LIN {X 0,Y 287.709,Z 666.106,A -85,B 0,C 180,E1 12553.998,E2 12553.998} C_VEL
LIN {X 0,Y 281.324,Z 683.017,A -85,B 0,C 180,E1 12550.975,E2 12550.975} C_VEL
LIN {X 0,Y 275.503,Z 697.991,A -85,B 0,C 180,E1 12547.706,E2 12547.706} C_VEL
LIN {X 0,Y 269.962,Z 712.115,A -85,B 0,C 180,E1 12543.941,E2 12543.941} C_VEL
LIN {X 0,Y 265.266,Z 724.533,A -85,B 0,C 180,E1 12539.897,E2 12539.897} C_VEL
LIN {X 0,Y 261.375,Z 735.692,A -85,B 0,C 180,E1 12535.368,E2 12535.368} C_VEL
LIN {X 0,Y 258.724,Z 744.628,A -85,B 0,C 180,E1 12530.826,E2 12530.826} C_VEL
LIN {X 0,Y 257.127,Z 751.706,A -85,B 0,C 180,E1 12526.164,E2 12526.164} C_VEL
LIN {X 0,Y 256.425,Z 757.033,A -85,B 0,C 180,E1 12521.47,E2 12521.47} C_VEL
LIN {X 0,Y 256.333,Z 760.365,A -85,B 0,C 180,E1 12517.17,E2 12517.17} C_VEL
LIN {X 0,Y 256.431,Z 762.152,A -85,B 0,C 180,E1 12513.129,E2 12513.129} C_VEL
LIN {X 0,Y 256.464,Z 762.649,A -85,B 0,C 180,E1 12509.106,E2 12509.106} C_VEL
LIN {X 0,Y 256.359,Z 761.883,A -85,B 0,C 180,E1 12505.077,E2 12505.077} C_VEL
LIN {X 0,Y 256.284,Z 759.711,A -85,B 0,C 180,E1 12500.764,E2 12500.764} C_VEL
LIN {X 0,Y 256.66,Z 755.693,A -85,B 0,C 180,E1 12496.023,E2 12496.023} C_VEL
LIN {X 0,Y 257.964,Z 749.671,A -85,B 0,C 180,E1 12491.036,E2 12491.036} C_VEL
LIN {X 0,Y 260.411,Z 741.966,A -85,B 0,C 180,E1 12486.224,E2 12486.224} C_VEL
LIN {X 0,Y 264.156,Z 732.301,A -85,B 0,C 180,E1 12481.515,E2 12481.515} C_VEL
LIN {X 0,Y 269.345,Z 720.5,A -85,B 0,C 180,E1 12476.928,E2 12476.928} C_VEL
LIN {X 0,Y 275.298,Z 707.685,A -85,B 0,C 180,E1 12472.922,E2 12472.922} C_VEL
LIN {X 0,Y 282.458,Z 692.507,A -85,B 0,C 180,E1 12469.09,E2 12469.09} C_VEL
LIN {X 0,Y 289.833,Z 676.554,A -85,B 0,C 180,E1 12465.824,E2 12465.824} C_VEL
LIN {X 0,Y 297.598,Z 658.888,A -85,B 0,C 180,E1 12462.909,E2 12462.909} C_VEL
LIN {X 0,Y 305.008,Z 640.783,A -85,B 0,C 180,E1 12460.488,E2 12460.488} C_VEL
LIN {X 0,Y 312.373,Z 620.899,A -85,B 0,C 180,E1 12458.352,E2 12458.352} C_VEL
LIN {X 0,Y 318.941,Z 600.695,A -85,B 0,C 180,E1 12456.626,E2 12456.626} C_VEL
LIN {X 0,Y 321.995,Z 590.5,A -85,B 0,C 180,E1 12455.859,E2 12455.859} C_VEL
LIN {X 0,Y 315.93,Z 596.748,A -85,B 0,C 180,E1 12455.169,E2 12455.169} C_VEL
LIN {X 0,Y 312.395,Z 600.249,A -85,B 0,C 180,E1 12454.729,E2 12454.729} C_VEL
LIN {X 0,Y 306.375,Z 605.854,A -85,B 0,C 180,E1 12453.921,E2 12453.921} C_VEL
LIN {X 0,Y 302.961,Z 608.865,A -85,B 0,C 180,E1 12453.445,E2 12453.445} C_VEL
LIN {X 0,Y 298.097,Z 612.903,A -85,B 0,C 180,E1 12452.684,E2 12452.684} C_VEL
LIN {X 0,Y 295.592,Z 614.826,A -85,B 0,C 180,E1 12452.259,E2 12452.259} C_VEL
LIN {X 0,Y 291.07,Z 618.329,A -85,B 0,C 180,E1 12451.475,E2 12451.475} C_VEL
LIN {X 0,Y 289.437,Z 619.438,A -85,B 0,C 180,E1 12451.094,E2 12451.094} C_VEL
LIN {X 0,Y 284.898,Z 632.295,A -85,B 0,C 180,E1 12448.737,E2 12448.737} C_VEL
LIN {X 0,Y 280.252,Z 644.016,A -85,B 0,C 180,E1 12446.028,E2 12446.028} C_VEL
LIN {X 0,Y 276.082,Z 653.459,A -85,B 0,C 180,E1 12443.25,E2 12443.25} C_VEL
LIN {X 0,Y 272.153,Z 661.429,A -85,B 0,C 180,E1 12440.202,E2 12440.202} C_VEL
LIN {X 0,Y 268.745,Z 667.609,A -85,B 0,C 180,E1 12437.026,E2 12437.026} C_VEL
LIN {X 0,Y 265.837,Z 672.016,A -85,B 0,C 180,E1 12433.706,E2 12433.706} C_VEL
LIN {X 0,Y 263.349,Z 674.833,A -85,B 0,C 180,E1 12430.057,E2 12430.057} C_VEL
LIN {X 0,Y 261.625,Z 675.693,A -85,B 0,C 180,E1 12426.583,E2 12426.583} C_VEL
LIN {X 0,Y 260.437,Z 674.815,A -85,B 0,C 180,E1 12423.08,E2 12423.08} C_VEL
LIN {X 0,Y 259.701,Z 672.036,A -85,B 0,C 180,E1 12419.337,E2 12419.337} C_VEL
LIN {X 0,Y 259.434,Z 667.616,A -85,B 0,C 180,E1 12415.8,E2 12415.8} C_VEL
LIN {X 0,Y 259.589,Z 661.3,A -85,B 0,C 180,E1 12412.252,E2 12412.252} C_VEL
LIN {X 0,Y 260.152,Z 653.545,A -85,B 0,C 180,E1 12408.92,E2 12408.92} C_VEL
LIN {X 0,Y 261.115,Z 643.862,A -85,B 0,C 180,E1 12405.648,E2 12405.648} C_VEL
LIN {X 0,Y 261.552,Z 640.556,A -85,B 0,C 180,E1 12404.592,E2 12404.592} C_VEL
LIN {X 0,Y 263.019,Z 640.91,A -85,B 0,C 180,E1 12403.661,E2 12403.661} C_VEL
LIN {X 0,Y 265.448,Z 640.458,A -85,B 0,C 180,E1 12402.688,E2 12402.688} C_VEL
LIN {X 0,Y 268.096,Z 640.355,A -85,B 0,C 180,E1 12401.517,E2 12401.517} C_VEL
LIN {X 0,Y 270.163,Z 640.044,A -85,B 0,C 180,E1 12400.768,E2 12400.768} C_VEL
LIN {X 0,Y 278.814,Z 638.787,A -85,B 0,C 180,E1 12397.88,E2 12397.88} C_VEL
LIN {X 0,Y 285.599,Z 637.414,A -85,B 0,C 180,E1 12396.039,E2 12396.039} C_VEL
LIN {X 0,Y 292.954,Z 635.796,A -85,B 0,C 180,E1 12394.312,E2 12394.312} C_VEL
LIN {X 0,Y 301.493,Z 633.669,A -85,B 0,C 180,E1 12392.603,E2 12392.603} C_VEL
LIN {X 0,Y 293.986,Z 648.836,A -85,B 0,C 180,E1 12389.754,E2 12389.754} C_VEL
LIN {X 0,Y 286.539,Z 662.886,A -85,B 0,C 180,E1 12386.51,E2 12386.51} C_VEL
LIN {X 0,Y 279.52,Z 675.51,A -85,B 0,C 180,E1 12382.91,E2 12382.91} C_VEL
LIN {X 0,Y 272.808,Z 687.29,A -85,B 0,C 180,E1 12378.707,E2 12378.707} C_VEL
LIN {X 0,Y 267.384,Z 696.902,A -85,B 0,C 180,E1 12374.369,E2 12374.369} C_VEL
LIN {X 0,Y 263.01,Z 704.996,A -85,B 0,C 180,E1 12369.693,E2 12369.693} C_VEL
LIN {X 0,Y 259.949,Z 711.213,A -85,B 0,C 180,E1 12364.968,E2 12364.968} C_VEL
LIN {X 0,Y 257.954,Z 715.929,A -85,B 0,C 180,E1 12360.002,E2 12360.002} C_VEL
LIN {X 0,Y 256.953,Z 718.932,A -85,B 0,C 180,E1 12355.097,E2 12355.097} C_VEL
LIN {X 0,Y 256.567,Z 720.347,A -85,B 0,C 180,E1 12350.533,E2 12350.533} C_VEL
LIN {X 0,Y 256.474,Z 720.34,A -85,B 0,C 180,E1 12346.302,E2 12346.302} C_VEL
LIN {X 0,Y 256.567,Z 719.146,A -85,B 0,C 180,E1 12341.92,E2 12341.92} C_VEL
LIN {X 0,Y 256.986,Z 716.554,A -85,B 0,C 180,E1 12337.377,E2 12337.377} C_VEL
LIN {X 0,Y 257.96,Z 712.498,A -85,B 0,C 180,E1 12332.889,E2 12332.889} C_VEL
LIN {X 0,Y 259.936,Z 706.41,A -85,B 0,C 180,E1 12328.016,E2 12328.016} C_VEL
LIN {X 0,Y 262.999,Z 698.454,A -85,B 0,C 180,E1 12323.232,E2 12323.232} C_VEL
LIN {X 0,Y 266.855,Z 689.477,A -85,B 0,C 180,E1 12318.984,E2 12318.984} C_VEL
LIN {X 0,Y 271.486,Z 679.247,A -85,B 0,C 180,E1 12315.061,E2 12315.061} C_VEL
LIN {X 0,Y 277.356,Z 666.333,A -85,B 0,C 180,E1 12311.068,E2 12311.068} C_VEL
LIN {X 0,Y 283.859,Z 651.692,A -85,B 0,C 180,E1 12307.422,E2 12307.422} C_VEL
LIN {X 0,Y 290.403,Z 636.19,A -85,B 0,C 180,E1 12304.29,E2 12304.29} C_VEL
LIN {X 0,Y 296.927,Z 619.534,A -85,B 0,C 180,E1 12301.544,E2 12301.544} C_VEL
LIN {X 0,Y 302.986,Z 602.453,A -85,B 0,C 180,E1 12299.236,E2 12299.236} C_VEL
LIN {X 0,Y 308.642,Z 584.487,A -85,B 0,C 180,E1 12297.248,E2 12297.248} C_VEL
LIN {X 0,Y 313.768,Z 565.683,A -85,B 0,C 180,E1 12295.555,E2 12295.555} C_VEL
LIN {X 0,Y 317.992,Z 547.266,A -85,B 0,C 180,E1 12294.209,E2 12294.209} C_VEL
LIN {X 0,Y 318.787,Z 543.221,A -85,B 0,C 180,E1 12293.959,E2 12293.959} C_VEL
LIN {X 0,Y 319.522,Z 537.124,A -85,B 0,C 180,E1 12293.495,E2 12293.495} C_VEL
LIN {X 0,Y 318.437,Z 518.424,A -85,B 0,C 180,E1 12291.694,E2 12291.694} C_VEL
LIN {X 0,Y 318.663,Z 511.085,A -85,B 0,C 180,E1 12291.25,E2 12291.25} C_VEL
LIN {X 0,Y 324.037,Z 467.251,A -85,B 0,C 180,E1 12289.77,E2 12289.77} C_VEL
LIN {X 0,Y 333.023,Z 393.238,A -85,B 0,C 180,E1 12287.708,E2 12287.708} C_VEL
LIN {X 0,Y 339.557,Z 329.299,A -85,B 0,C 180,E1 12286.143,E2 12286.143} C_VEL
LIN {X 0,Y 330.547,Z 317.786,A -85,B 0,C 180,E1 12283.128,E2 12283.128} C_VEL
LIN {X 0,Y 322.358,Z 308.216,A -85,B 0,C 180,E1 12280.12,E2 12280.12} C_VEL
LIN {X 0,Y 315.707,Z 301.17,A -85,B 0,C 180,E1 12277.388,E2 12277.388} C_VEL
LIN {X 0,Y 311.912,Z 297.367,A -85,B 0,C 180,E1 12275.692,E2 12275.692} C_VEL
LIN {X 0,Y 307.01,Z 292.557,A -85,B 0,C 180,E1 12273.283,E2 12273.283} C_VEL
LIN {X 0,Y 300.753,Z 286.807,A -85,B 0,C 180,E1 12269.694,E2 12269.694} C_VEL
LIN {X 0,Y 298.843,Z 282.267,A -85,B 0,C 180,E1 12262.215,E2 12262.215} C_VEL
LIN {X 0,Y 298.718,Z 282.233,A -85,B 0,C 180,E1 12256.13,E2 12256.13} C_VEL
LIN {X 0,Y 298.885,Z 283.132,A -85,B 0,C 180,E1 12253.938,E2 12253.938} C_VEL
LIN {X 0,Y 300.939,Z 287.174,A -85,B 0,C 180,E1 12247.638,E2 12247.638} C_VEL
LIN {X 0,Y 303.087,Z 291.944,A -85,B 0,C 180,E1 12243.405,E2 12243.405} C_VEL
LIN {X 0,Y 305.298,Z 296.953,A -85,B 0,C 180,E1 12240.001,E2 12240.001} C_VEL
LIN {X 0,Y 308.334,Z 303.509,A -85,B 0,C 180,E1 12236.282,E2 12236.282} C_VEL
LIN {X 0,Y 311.872,Z 311.892,A -85,B 0,C 180,E1 12232.447,E2 12232.447} C_VEL
LIN {X 0,Y 315.856,Z 321.763,A -85,B 0,C 180,E1 12228.682,E2 12228.682} C_VEL
LIN {X 0,Y 320.085,Z 333.219,A -85,B 0,C 180,E1 12224.974,E2 12224.974} C_VEL
LIN {X 0,Y 324.216,Z 345.387,A -85,B 0,C 180,E1 12221.596,E2 12221.596} C_VEL
LIN {X 0,Y 318.081,Z 372.788,A -85,B 0,C 180,E1 12218.422,E2 12218.422} C_VEL
LIN {X 0,Y 316.025,Z 387.195,A -85,B 0,C 180,E1 12216.606,E2 12216.606} C_VEL
LIN {X 0,Y 319.632,Z 409.436,A -85,B 0,C 180,E1 12214.513,E2 12214.513} C_VEL
LIN {X 0,Y 324.829,Z 432.239,A -85,B 0,C 180,E1 12212.129,E2 12212.129} C_VEL
LIN {X 0,Y 331.021,Z 453.159,A -85,B 0,C 180,E1 12209.682,E2 12209.682} C_VEL
LIN {X 0,Y 333.918,Z 461.741,A -85,B 0,C 180,E1 12208.622,E2 12208.622} C_VEL
LIN {X 0,Y 329.325,Z 485.74,A -85,B 0,C 180,E1 12208.295,E2 12208.295} C_VEL
LIN {X 0,Y 325.309,Z 507.365,A -85,B 0,C 180,E1 12207.685,E2 12207.685} C_VEL
LIN {X 0,Y 319.116,Z 537.78,A -85,B 0,C 180,E1 12206.453,E2 12206.453} C_VEL
LIN {X 0,Y 312.613,Z 564.487,A -85,B 0,C 180,E1 12205.075,E2 12205.075} C_VEL
LIN {X 0,Y 305.507,Z 591.109,A -85,B 0,C 180,E1 12203.305,E2 12203.305} C_VEL
LIN {X 0,Y 298.545,Z 615.325,A -85,B 0,C 180,E1 12201.292,E2 12201.292} C_VEL
LIN {X 0,Y 292.302,Z 634.979,A -85,B 0,C 180,E1 12199.244,E2 12199.244} C_VEL
LIN {X 0,Y 285.775,Z 653.697,A -85,B 0,C 180,E1 12196.843,E2 12196.843} C_VEL
LIN {X 0,Y 279.285,Z 670.834,A -85,B 0,C 180,E1 12194.132,E2 12194.132} C_VEL
LIN {X 0,Y 272.764,Z 687.205,A -85,B 0,C 180,E1 12190.965,E2 12190.965} C_VEL
LIN {X 0,Y 266.949,Z 701.43,A -85,B 0,C 180,E1 12187.627,E2 12187.627} C_VEL
LIN {X 0,Y 261.357,Z 715.082,A -85,B 0,C 180,E1 12183.691,E2 12183.691} C_VEL
LIN {X 0,Y 256.61,Z 727.181,A -85,B 0,C 180,E1 12179.403,E2 12179.403} C_VEL
LIN {X 0,Y 253.037,Z 737.149,A -85,B 0,C 180,E1 12175.011,E2 12175.011} C_VEL
LIN {X 0,Y 250.368,Z 746.008,A -85,B 0,C 180,E1 12170.087,E2 12170.087} C_VEL
LIN {X 0,Y 248.944,Z 752.544,A -85,B 0,C 180,E1 12165.371,E2 12165.371} C_VEL
LIN {X 0,Y 248.392,Z 757.273,A -85,B 0,C 180,E1 12160.67,E2 12160.67} C_VEL
LIN {X 0,Y 248.376,Z 760.301,A -85,B 0,C 180,E1 12156.117,E2 12156.117} C_VEL
LIN {X 0,Y 248.488,Z 761.748,A -85,B 0,C 180,E1 12151.844,E2 12151.844} C_VEL
LIN {X 0,Y 248.469,Z 761.881,A -85,B 0,C 180,E1 12147.924,E2 12147.924} C_VEL
LIN {X 0,Y 248.334,Z 760.797,A -85,B 0,C 180,E1 12143.759,E2 12143.759} C_VEL
LIN {X 0,Y 248.351,Z 758.132,A -85,B 0,C 180,E1 12139.092,E2 12139.092} C_VEL
LIN {X 0,Y 249.007,Z 753.673,A -85,B 0,C 180,E1 12134.154,E2 12134.154} C_VEL
LIN {X 0,Y 250.699,Z 747.449,A -85,B 0,C 180,E1 12129.209,E2 12129.209} C_VEL
LIN {X 0,Y 253.66,Z 739.35,A -85,B 0,C 180,E1 12124.304,E2 12124.304} C_VEL
LIN {X 0,Y 258.05,Z 729.293,A -85,B 0,C 180,E1 12119.497,E2 12119.497} C_VEL
LIN {X 0,Y 263.636,Z 717.634,A -85,B 0,C 180,E1 12115.062,E2 12115.062} C_VEL
LIN {X 0,Y 270.591,Z 703.684,A -85,B 0,C 180,E1 12110.812,E2 12110.812} C_VEL
LIN {X 0,Y 277.989,Z 688.837,A -85,B 0,C 180,E1 12107.172,E2 12107.172} C_VEL
LIN {X 0,Y 285.835,Z 672.631,A -85,B 0,C 180,E1 12103.969,E2 12103.969} C_VEL
LIN {X 0,Y 293.702,Z 655.348,A -85,B 0,C 180,E1 12101.204,E2 12101.204} C_VEL
LIN {X 0,Y 301.822,Z 636.092,A -85,B 0,C 180,E1 12098.725,E2 12098.725} C_VEL
LIN {X 0,Y 309.274,Z 616.271,A -85,B 0,C 180,E1 12096.7,E2 12096.7} C_VEL
LIN {X 0,Y 312.818,Z 605.818,A -85,B 0,C 180,E1 12095.797,E2 12095.797} C_VEL
LIN {X 0,Y 306.207,Z 611.634,A -85,B 0,C 180,E1 12094.955,E2 12094.955} C_VEL
LIN {X 0,Y 298.851,Z 617.69,A -85,B 0,C 180,E1 12093.967,E2 12093.967} C_VEL
LIN {X 0,Y 293.954,Z 621.35,A -85,B 0,C 180,E1 12093.204,E2 12093.204} C_VEL
LIN {X 0,Y 288.566,Z 625.001,A -85,B 0,C 180,E1 12092.248,E2 12092.248} C_VEL
LIN {X 0,Y 283.885,Z 628.269,A -85,B 0,C 180,E1 12091.416,E2 12091.416} C_VEL
LIN {X 0,Y 281.615,Z 629.73,A -85,B 0,C 180,E1 12090.866,E2 12090.866} C_VEL
LIN {X 0,Y 276.211,Z 642.527,A -85,B 0,C 180,E1 12088.072,E2 12088.072} C_VEL
LIN {X 0,Y 271.175,Z 653.092,A -85,B 0,C 180,E1 12085.088,E2 12085.088} C_VEL
LIN {X 0,Y 266.745,Z 661.49,A -85,B 0,C 180,E1 12082.013,E2 12082.013} C_VEL
LIN {X 0,Y 262.661,Z 668.241,A -85,B 0,C 180,E1 12078.648,E2 12078.648} C_VEL
LIN {X 0,Y 259.286,Z 673.072,A -85,B 0,C 180,E1 12075.201,E2 12075.201} C_VEL
LIN {X 0,Y 256.551,Z 676.036,A -85,B 0,C 180,E1 12071.692,E2 12071.692} C_VEL
LIN {X 0,Y 254.351,Z 677.274,A -85,B 0,C 180,E1 12067.907,E2 12067.907} C_VEL
LIN {X 0,Y 252.909,Z 676.728,A -85,B 0,C 180,E1 12064.307,E2 12064.307} C_VEL
LIN {X 0,Y 251.98,Z 674.352,A -85,B 0,C 180,E1 12060.585,E2 12060.585} C_VEL
LIN {X 0,Y 251.529,Z 670.008,A -85,B 0,C 180,E1 12056.73,E2 12056.73} C_VEL
LIN {X 0,Y 251.566,Z 664.192,A -85,B 0,C 180,E1 12053.151,E2 12053.151} C_VEL
LIN {X 0,Y 252.063,Z 656.173,A -85,B 0,C 180,E1 12049.486,E2 12049.486} C_VEL
LIN {X 0,Y 253,Z 646.667,A -85,B 0,C 180,E1 12046.049,E2 12046.049} C_VEL
LIN {X 0,Y 254.434,Z 647.022,A -85,B 0,C 180,E1 12044.967,E2 12044.967} C_VEL
LIN {X 0,Y 256.654,Z 646.641,A -85,B 0,C 180,E1 12043.942,E2 12043.942} C_VEL
LIN {X 0,Y 259.072,Z 646.592,A -85,B 0,C 180,E1 12042.711,E2 12042.711} C_VEL
LIN {X 0,Y 260.951,Z 646.353,A -85,B 0,C 180,E1 12041.918,E2 12041.918} C_VEL
LIN {X 0,Y 269.062,Z 645.407,A -85,B 0,C 180,E1 12038.867,E2 12038.867} C_VEL
LIN {X 0,Y 275.424,Z 644.367,A -85,B 0,C 180,E1 12036.916,E2 12036.916} C_VEL
LIN {X 0,Y 282.085,Z 643.093,A -85,B 0,C 180,E1 12035.15,E2 12035.15} C_VEL
LIN {X 0,Y 289.926,Z 641.408,A -85,B 0,C 180,E1 12033.363,E2 12033.363} C_VEL
LIN {X 0,Y 293.134,Z 640.746,A -85,B 0,C 180,E1 12032.68,E2 12032.68} C_VEL
LIN {X 0,Y 285.157,Z 655.655,A -85,B 0,C 180,E1 12029.606,E2 12029.606} C_VEL
LIN {X 0,Y 277.118,Z 669.729,A -85,B 0,C 180,E1 12025.995,E2 12025.995} C_VEL
LIN {X 0,Y 269.767,Z 682.054,A -85,B 0,C 180,E1 12022.028,E2 12022.028} C_VEL
LIN {X 0,Y 263.383,Z 692.576,A -85,B 0,C 180,E1 12017.754,E2 12017.754} C_VEL
LIN {X 0,Y 258.195,Z 701.295,A -85,B 0,C 180,E1 12013.27,E2 12013.27} C_VEL
LIN {X 0,Y 254.094,Z 708.56,A -85,B 0,C 180,E1 12008.443,E2 12008.443} C_VEL
LIN {X 0,Y 251.183,Z 714.311,A -85,B 0,C 180,E1 12003.286,E2 12003.286} C_VEL
LIN {X 0,Y 249.532,Z 718.225,A -85,B 0,C 180,E1 11998.171,E2 11998.171} C_VEL
LIN {X 0,Y 248.8,Z 720.404,A -85,B 0,C 180,E1 11993.445,E2 11993.445} C_VEL
LIN {X 0,Y 248.533,Z 721.128,A -85,B 0,C 180,E1 11989.016,E2 11989.016} C_VEL
LIN {X 0,Y 248.517,Z 720.638,A -85,B 0,C 180,E1 11984.445,E2 11984.445} C_VEL
LIN {X 0,Y 248.718,Z 718.924,A -85,B 0,C 180,E1 11979.955,E2 11979.955} C_VEL
LIN {X 0,Y 249.382,Z 715.683,A -85,B 0,C 180,E1 11975.291,E2 11975.291} C_VEL
LIN {X 0,Y 250.828,Z 710.804,A -85,B 0,C 180,E1 11970.457,E2 11970.457} C_VEL
LIN {X 0,Y 253.255,Z 704.306,A -85,B 0,C 180,E1 11965.698,E2 11965.698} C_VEL
LIN {X 0,Y 256.787,Z 696.065,A -85,B 0,C 180,E1 11961.04,E2 11961.04} C_VEL
LIN {X 0,Y 261.249,Z 686.421,A -85,B 0,C 180,E1 11956.725,E2 11956.725} C_VEL
LIN {X 0,Y 266.764,Z 674.755,A -85,B 0,C 180,E1 11952.552,E2 11952.552} C_VEL
LIN {X 0,Y 272.638,Z 662.275,A -85,B 0,C 180,E1 11948.937,E2 11948.937} C_VEL
LIN {X 0,Y 278.937,Z 648.484,A -85,B 0,C 180,E1 11945.656,E2 11945.656} C_VEL
LIN {X 0,Y 285.698,Z 632.79,A -85,B 0,C 180,E1 11942.6,E2 11942.6} C_VEL
LIN {X 0,Y 292.354,Z 615.994,A -85,B 0,C 180,E1 11939.932,E2 11939.932} C_VEL
LIN {X 0,Y 298.494,Z 598.888,A -85,B 0,C 180,E1 11937.706,E2 11937.706} C_VEL
LIN {X 0,Y 304.165,Z 581.035,A -85,B 0,C 180,E1 11935.798,E2 11935.798} C_VEL
LIN {X 0,Y 309.49,Z 561.333,A -85,B 0,C 180,E1 11934.101,E2 11934.101} C_VEL
LIN {X 0,Y 313.859,Z 541.499,A -85,B 0,C 180,E1 11932.751,E2 11932.751} C_VEL
LIN {X 0,Y 317.269,Z 521.59,A -85,B 0,C 180,E1 11931.701,E2 11931.701} C_VEL
LIN {X 0,Y 318.663,Z 511.085,A -85,B 0,C 180,E1 11931.25,E2 11931.25} C_VEL
LIN {X 0,Y 318.93,Z 503.689,A -85,B 0,C 180,E1 11930.826,E2 11930.826} C_VEL
LIN {X 0,Y 317.385,Z 484.34,A -85,B 0,C 180,E1 11929.284,E2 11929.284} C_VEL
LIN {X 0,Y 317.734,Z 477.943,A -85,B 0,C 180,E1 11928.968,E2 11928.968} C_VEL
LIN {X 0,Y 327.089,Z 405.309,A -85,B 0,C 180,E1 11926.876,E2 11926.876} C_VEL
LIN {X 0,Y 334.404,Z 338.419,A -85,B 0,C 180,E1 11925.22,E2 11925.22} C_VEL
LIN {X 0,Y 334.711,Z 333.682,A -85,B 0,C 180,E1 11925.071,E2 11925.071} C_VEL
LIN {X 0,Y 324.797,Z 321.044,A -85,B 0,C 180,E1 11921.56,E2 11921.56} C_VEL
LIN {X 0,Y 316.095,Z 311.142,A -85,B 0,C 180,E1 11918.085,E2 11918.085} C_VEL
LIN {X 0,Y 310.031,Z 304.952,A -85,B 0,C 180,E1 11915.373,E2 11915.373} C_VEL
LIN {X 0,Y 305.207,Z 300.156,A -85,B 0,C 180,E1 11912.945,E2 11912.945} C_VEL
LIN {X 0,Y 298.864,Z 294.412,A -85,B 0,C 180,E1 11909.239,E2 11909.239} C_VEL
LIN {X 0,Y 295.589,Z 292.119,A -85,B 0,C 180,E1 11906.954,E2 11906.954} C_VEL
LIN {X 0,Y 294.925,Z 289.241,A -85,B 0,C 180,E1 11902.106,E2 11902.106} C_VEL
LIN {X 0,Y 294.817,Z 289.216,A -85,B 0,C 180,E1 11896.148,E2 11896.148} C_VEL
LIN {X 0,Y 294.962,Z 290.165,A -85,B 0,C 180,E1 11893.927,E2 11893.927} C_VEL
LIN {X 0,Y 296.908,Z 294.121,A -85,B 0,C 180,E1 11887.742,E2 11887.742} C_VEL
LIN {X 0,Y 298.993,Z 298.946,A -85,B 0,C 180,E1 11883.452,E2 11883.452} C_VEL
LIN {X 0,Y 301.055,Z 303.683,A -85,B 0,C 180,E1 11880.191,E2 11880.191} C_VEL
LIN {X 0,Y 303.85,Z 309.92,A -85,B 0,C 180,E1 11876.605,E2 11876.605} C_VEL
LIN {X 0,Y 307.296,Z 318.329,A -85,B 0,C 180,E1 11872.71,E2 11872.71} C_VEL
LIN {X 0,Y 310.971,Z 327.744,A -85,B 0,C 180,E1 11869.065,E2 11869.065} C_VEL
LIN {X 0,Y 315.084,Z 339.249,A -85,B 0,C 180,E1 11865.294,E2 11865.294} C_VEL
LIN {X 0,Y 318.412,Z 349.715,A -85,B 0,C 180,E1 11862.361,E2 11862.361} C_VEL
LIN {X 0,Y 312.275,Z 376.379,A -85,B 0,C 180,E1 11859.218,E2 11859.218} C_VEL
LIN {X 0,Y 311.243,Z 383.393,A -85,B 0,C 180,E1 11858.357,E2 11858.357} C_VEL
LIN {X 0,Y 314.553,Z 407.697,A -85,B 0,C 180,E1 11856.104,E2 11856.104} C_VEL
LIN {X 0,Y 319.175,Z 430.509,A -85,B 0,C 180,E1 11853.738,E2 11853.738} C_VEL
LIN {X 0,Y 325.029,Z 452.707,A -85,B 0,C 180,E1 11851.147,E2 11851.147} C_VEL
LIN {X 0,Y 328.515,Z 464.338,A -85,B 0,C 180,E1 11849.705,E2 11849.705} C_VEL
LIN {X 0,Y 323.381,Z 490.681,A -85,B 0,C 180,E1 11849.287,E2 11849.287} C_VEL
LIN {X 0,Y 318.896,Z 514.316,A -85,B 0,C 180,E1 11848.52,E2 11848.52} C_VEL
LIN {X 0,Y 312.309,Z 543.991,A -85,B 0,C 180,E1 11847.245,E2 11847.245} C_VEL
LIN {X 0,Y 305.733,Z 569.916,A -85,B 0,C 180,E1 11845.832,E2 11845.832} C_VEL
LIN {X 0,Y 298.532,Z 595.679,A -85,B 0,C 180,E1 11844.034,E2 11844.034} C_VEL
LIN {X 0,Y 291.098,Z 620.431,A -85,B 0,C 180,E1 11841.865,E2 11841.865} C_VEL
LIN {X 0,Y 284.741,Z 639.238,A -85,B 0,C 180,E1 11839.779,E2 11839.779} C_VEL
LIN {X 0,Y 277.839,Z 657.811,A -85,B 0,C 180,E1 11837.234,E2 11837.234} C_VEL
LIN {X 0,Y 271.013,Z 674.974,A -85,B 0,C 180,E1 11834.342,E2 11834.342} C_VEL
LIN {X 0,Y 264.102,Z 691.372,A -85,B 0,C 180,E1 11830.916,E2 11830.916} C_VEL
LIN {X 0,Y 257.895,Z 705.812,A -85,B 0,C 180,E1 11827.215,E2 11827.215} C_VEL
LIN {X 0,Y 252.393,Z 718.669,A -85,B 0,C 180,E1 11823.14,E2 11823.14} C_VEL
LIN {X 0,Y 247.785,Z 730.049,A -85,B 0,C 180,E1 11818.697,E2 11818.697} C_VEL
LIN {X 0,Y 244.392,Z 739.423,A -85,B 0,C 180,E1 11814.149,E2 11814.149} C_VEL
LIN {X 0,Y 242.03,Z 747.265,A -85,B 0,C 180,E1 11809.298,E2 11809.298} C_VEL
LIN {X 0,Y 240.776,Z 753.313,A -85,B 0,C 180,E1 11804.427,E2 11804.427} C_VEL
LIN {X 0,Y 240.367,Z 757.646,A -85,B 0,C 180,E1 11799.578,E2 11799.578} C_VEL
LIN {X 0,Y 240.436,Z 760.186,A -85,B 0,C 180,E1 11795.01,E2 11795.01} C_VEL
LIN {X 0,Y 240.526,Z 761.258,A -85,B 0,C 180,E1 11790.714,E2 11790.714} C_VEL
LIN {X 0,Y 240.445,Z 761.047,A -85,B 0,C 180,E1 11786.423,E2 11786.423} C_VEL
LIN {X 0,Y 240.308,Z 759.449,A -85,B 0,C 180,E1 11781.867,E2 11781.867} C_VEL
LIN {X 0,Y 240.524,Z 756.253,A -85,B 0,C 180,E1 11777.027,E2 11777.027} C_VEL
LIN {X 0,Y 241.605,Z 751.238,A -85,B 0,C 180,E1 11771.917,E2 11771.917} C_VEL
LIN {X 0,Y 244.042,Z 744.096,A -85,B 0,C 180,E1 11766.583,E2 11766.583} C_VEL
LIN {X 0,Y 247.809,Z 735.331,A -85,B 0,C 180,E1 11761.568,E2 11761.568} C_VEL
LIN {X 0,Y 253.117,Z 724.493,A -85,B 0,C 180,E1 11756.696,E2 11756.696} C_VEL
LIN {X 0,Y 259.635,Z 712.078,A -85,B 0,C 180,E1 11752.243,E2 11752.243} C_VEL
LIN {X 0,Y 267.115,Z 697.993,A -85,B 0,C 180,E1 11748.218,E2 11748.218} C_VEL
LIN {X 0,Y 274.838,Z 683.232,A -85,B 0,C 180,E1 11744.813,E2 11744.813} C_VEL
LIN {X 0,Y 283.481,Z 665.962,A -85,B 0,C 180,E1 11741.604,E2 11741.604} C_VEL
LIN {X 0,Y 291.826,Z 648.029,A -85,B 0,C 180,E1 11738.944,E2 11738.944} C_VEL
LIN {X 0,Y 299.886,Z 629.029,A -85,B 0,C 180,E1 11736.691,E2 11736.691} C_VEL
LIN {X 0,Y 303.591,Z 619.39,A -85,B 0,C 180,E1 11735.721,E2 11735.721} C_VEL
LIN {X 0,Y 297.258,Z 624.134,A -85,B 0,C 180,E1 11734.876,E2 11734.876} C_VEL
LIN {X 0,Y 288.924,Z 629.899,A -85,B 0,C 180,E1 11733.621,E2 11733.621} C_VEL
LIN {X 0,Y 281.159,Z 634.752,A -85,B 0,C 180,E1 11732.237,E2 11732.237} C_VEL
LIN {X 0,Y 274.569,Z 638.458,A -85,B 0,C 180,E1 11730.894,E2 11730.894} C_VEL
LIN {X 0,Y 273.687,Z 639.057,A -85,B 0,C 180,E1 11730.639,E2 11730.639} C_VEL
LIN {X 0,Y 268.477,Z 649.505,A -85,B 0,C 180,E1 11727.985,E2 11727.985} C_VEL
LIN {X 0,Y 263.27,Z 658.88,A -85,B 0,C 180,E1 11724.932,E2 11724.932} C_VEL
LIN {X 0,Y 258.714,Z 666.293,A -85,B 0,C 180,E1 11721.777,E2 11721.777} C_VEL
LIN {X 0,Y 254.533,Z 672.146,A -85,B 0,C 180,E1 11718.315,E2 11718.315} C_VEL
LIN {X 0,Y 250.905,Z 676.362,A -85,B 0,C 180,E1 11714.539,E2 11714.539} C_VEL
LIN {X 0,Y 248.185,Z 678.481,A -85,B 0,C 180,E1 11710.914,E2 11710.914} C_VEL
LIN {X 0,Y 246.051,Z 678.876,A -85,B 0,C 180,E1 11707.002,E2 11707.002} C_VEL
LIN {X 0,Y 244.692,Z 677.527,A -85,B 0,C 180,E1 11703.279,E2 11703.279} C_VEL
LIN {X 0,Y 243.883,Z 674.454,A -85,B 0,C 180,E1 11699.529,E2 11699.529} C_VEL
LIN {X 0,Y 243.555,Z 669.614,A -85,B 0,C 180,E1 11695.761,E2 11695.761} C_VEL
LIN {X 0,Y 243.716,Z 662.917,A -85,B 0,C 180,E1 11691.981,E2 11691.981} C_VEL
LIN {X 0,Y 244.329,Z 654.683,A -85,B 0,C 180,E1 11688.432,E2 11688.432} C_VEL
LIN {X 0,Y 244.551,Z 652.561,A -85,B 0,C 180,E1 11687.604,E2 11687.604} C_VEL
LIN {X 0,Y 246.017,Z 652.894,A -85,B 0,C 180,E1 11686.365,E2 11686.365} C_VEL
LIN {X 0,Y 247.738,Z 652.568,A -85,B 0,C 180,E1 11685.508,E2 11685.508} C_VEL
LIN {X 0,Y 250.278,Z 652.631,A -85,B 0,C 180,E1 11683.998,E2 11683.998} C_VEL
LIN {X 0,Y 252.339,Z 652.473,A -85,B 0,C 180,E1 11682.949,E2 11682.949} C_VEL
LIN {X 0,Y 259.423,Z 651.666,A -85,B 0,C 180,E1 11679.938,E2 11679.938} C_VEL
LIN {X 0,Y 270.603,Z 650.09,A -85,B 0,C 180,E1 11676.249,E2 11676.249} C_VEL
LIN {X 0,Y 284.26,Z 647.451,A -85,B 0,C 180,E1 11672.862,E2 11672.862} C_VEL
LIN {X 0,Y 284.704,Z 647.341,A -85,B 0,C 180,E1 11672.772,E2 11672.772} C_VEL
LIN {X 0,Y 276.598,Z 661.462,A -85,B 0,C 180,E1 11669.596,E2 11669.596} C_VEL
LIN {X 0,Y 268.827,Z 674.201,A -85,B 0,C 180,E1 11666.039,E2 11666.039} C_VEL
LIN {X 0,Y 261.439,Z 685.826,A -85,B 0,C 180,E1 11661.984,E2 11661.984} C_VEL
LIN {X 0,Y 254.924,Z 695.969,A -85,B 0,C 180,E1 11657.509,E2 11657.509} C_VEL
LIN {X 0,Y 249.767,Z 704.169,A -85,B 0,C 180,E1 11652.886,E2 11652.886} C_VEL
LIN {X 0,Y 245.707,Z 711.01,A -85,B 0,C 180,E1 11647.865,E2 11647.865} C_VEL
LIN {X 0,Y 242.95,Z 716.21,A -85,B 0,C 180,E1 11642.625,E2 11642.625} C_VEL
LIN {X 0,Y 241.402,Z 719.638,A -85,B 0,C 180,E1 11637.371,E2 11637.371} C_VEL
LIN {X 0,Y 240.749,Z 721.379,A -85,B 0,C 180,E1 11632.463,E2 11632.463} C_VEL
LIN {X 0,Y 240.535,Z 721.787,A -85,B 0,C 180,E1 11627.665,E2 11627.665} C_VEL
LIN {X 0,Y 240.575,Z 720.947,A -85,B 0,C 180,E1 11623.214,E2 11623.214} C_VEL
LIN {X 0,Y 240.907,Z 718.678,A -85,B 0,C 180,E1 11618.353,E2 11618.353} C_VEL
LIN {X 0,Y 241.894,Z 714.836,A -85,B 0,C 180,E1 11613.318,E2 11613.318} C_VEL
LIN {X 0,Y 243.769,Z 709.438,A -85,B 0,C 180,E1 11608.355,E2 11608.355} C_VEL
LIN {X 0,Y 246.907,Z 701.953,A -85,B 0,C 180,E1 11603.256,E2 11603.256} C_VEL
LIN {X 0,Y 251.119,Z 692.917,A -85,B 0,C 180,E1 11598.517,E2 11598.517} C_VEL
LIN {X 0,Y 256.269,Z 682.42,A -85,B 0,C 180,E1 11594.151,E2 11594.151} C_VEL
LIN {X 0,Y 262.18,Z 670.509,A -85,B 0,C 180,E1 11590.159,E2 11590.159} C_VEL
LIN {X 0,Y 268.671,Z 657.159,A -85,B 0,C 180,E1 11586.535,E2 11586.535} C_VEL
LIN {X 0,Y 275.532,Z 642.348,A -85,B 0,C 180,E1 11583.258,E2 11583.258} C_VEL
LIN {X 0,Y 282.383,Z 626.518,A -85,B 0,C 180,E1 11580.4,E2 11580.4} C_VEL
LIN {X 0,Y 288.777,Z 610.432,A -85,B 0,C 180,E1 11578.012,E2 11578.012} C_VEL
LIN {X 0,Y 294.986,Z 592.943,A -85,B 0,C 180,E1 11575.878,E2 11575.878} C_VEL
LIN {X 0,Y 300.906,Z 573.621,A -85,B 0,C 180,E1 11573.975,E2 11573.975} C_VEL
LIN {X 0,Y 305.893,Z 554.109,A -85,B 0,C 180,E1 11572.439,E2 11572.439} C_VEL
LIN {X 0,Y 309.872,Z 534.895,A -85,B 0,C 180,E1 11571.246,E2 11571.246} C_VEL
LIN {X 0,Y 313.107,Z 514.369,A -85,B 0,C 180,E1 11570.263,E2 11570.263} C_VEL
LIN {X 0,Y 317.734,Z 477.943,A -85,B 0,C 180,E1 11568.968,E2 11568.968} C_VEL
LIN {X 0,Y 318.134,Z 470.477,A -85,B 0,C 180,E1 11568.586,E2 11568.586} C_VEL
LIN {X 0,Y 317.122,Z 450.95,A -85,B 0,C 180,E1 11567.088,E2 11567.088} C_VEL
LIN {X 0,Y 317.568,Z 444.518,A -85,B 0,C 180,E1 11566.79,E2 11566.79} C_VEL
LIN {X 0,Y 326.106,Z 376.251,A -85,B 0,C 180,E1 11564.953,E2 11564.953} C_VEL
LIN {X 0,Y 330.11,Z 338.452,A -85,B 0,C 180,E1 11564.035,E2 11564.035} C_VEL
LIN {X 0,Y 321.697,Z 327.645,A -85,B 0,C 180,E1 11560.923,E2 11560.923} C_VEL
LIN {X 0,Y 313.932,Z 318.547,A -85,B 0,C 180,E1 11557.7,E2 11557.7} C_VEL
LIN {X 0,Y 307.787,Z 312.187,A -85,B 0,C 180,E1 11554.873,E2 11554.873} C_VEL
LIN {X 0,Y 303.243,Z 307.628,A -85,B 0,C 180,E1 11552.511,E2 11552.511} C_VEL
LIN {X 0,Y 297.324,Z 302.157,A -85,B 0,C 180,E1 11548.964,E2 11548.964} C_VEL
LIN {X 0,Y 291.101,Z 297.33,A -85,B 0,C 180,E1 11544.126,E2 11544.126} C_VEL
LIN {X 0,Y 290.966,Z 296.194,A -85,B 0,C 180,E1 11541.786,E2 11541.786} C_VEL
LIN {X 0,Y 290.973,Z 296.253,A -85,B 0,C 180,E1 11535.814,E2 11535.814} C_VEL
LIN {X 0,Y 292.839,Z 300.834,A -85,B 0,C 180,E1 11528.043,E2 11528.043} C_VEL
LIN {X 0,Y 294.816,Z 305.657,A -85,B 0,C 180,E1 11523.695,E2 11523.695} C_VEL
LIN {X 0,Y 296.702,Z 310.099,A -85,B 0,C 180,E1 11520.58,E2 11520.58} C_VEL
LIN {X 0,Y 299.387,Z 316.346,A -85,B 0,C 180,E1 11516.93,E2 11516.93} C_VEL
LIN {X 0,Y 302.566,Z 324.32,A -85,B 0,C 180,E1 11513.168,E2 11513.168} C_VEL
LIN {X 0,Y 306.101,Z 333.725,A -85,B 0,C 180,E1 11509.461,E2 11509.461} C_VEL
LIN {X 0,Y 310.093,Z 345.282,A -85,B 0,C 180,E1 11505.625,E2 11505.625} C_VEL
LIN {X 0,Y 312.677,Z 353.904,A -85,B 0,C 180,E1 11503.169,E2 11503.169} C_VEL
LIN {X 0,Y 306.795,Z 379.34,A -85,B 0,C 180,E1 11500.151,E2 11500.151} C_VEL
LIN {X 0,Y 309.526,Z 404.098,A -85,B 0,C 180,E1 11497.907,E2 11497.907} C_VEL
LIN {X 0,Y 313.499,Z 427.252,A -85,B 0,C 180,E1 11495.531,E2 11495.531} C_VEL
LIN {X 0,Y 318.427,Z 448.942,A -85,B 0,C 180,E1 11493.043,E2 11493.043} C_VEL
LIN {X 0,Y 323.269,Z 466.796,A -85,B 0,C 180,E1 11490.817,E2 11490.817} C_VEL
LIN {X 0,Y 317.965,Z 493.165,A -85,B 0,C 180,E1 11490.351,E2 11490.351} C_VEL
LIN {X 0,Y 312.859,Z 519.062,A -85,B 0,C 180,E1 11489.456,E2 11489.456} C_VEL
LIN {X 0,Y 306.258,Z 547.401,A -85,B 0,C 180,E1 11488.203,E2 11488.203} C_VEL
LIN {X 0,Y 299.131,Z 574.141,A -85,B 0,C 180,E1 11486.682,E2 11486.682} C_VEL
LIN {X 0,Y 291.428,Z 600.831,A -85,B 0,C 180,E1 11484.741,E2 11484.741} C_VEL
LIN {X 0,Y 284.615,Z 622.385,A -85,B 0,C 180,E1 11482.765,E2 11482.765} C_VEL
LIN {X 0,Y 277.768,Z 641.753,A -85,B 0,C 180,E1 11480.544,E2 11480.544} C_VEL
LIN {X 0,Y 270.925,Z 659.364,A -85,B 0,C 180,E1 11478.042,E2 11478.042} C_VEL
LIN {X 0,Y 263.687,Z 676.59,A -85,B 0,C 180,E1 11475.006,E2 11475.006} C_VEL
LIN {X 0,Y 256.823,Z 692.208,A -85,B 0,C 180,E1 11471.628,E2 11471.628} C_VEL
LIN {X 0,Y 250.536,Z 706.113,A -85,B 0,C 180,E1 11467.922,E2 11467.922} C_VEL
LIN {X 0,Y 244.493,Z 719.617,A -85,B 0,C 180,E1 11463.462,E2 11463.462} C_VEL
LIN {X 0,Y 239.774,Z 730.746,A -85,B 0,C 180,E1 11458.873,E2 11458.873} C_VEL
LIN {X 0,Y 236.135,Z 740.382,A -85,B 0,C 180,E1 11453.852,E2 11453.852} C_VEL
LIN {X 0,Y 233.807,Z 748.117,A -85,B 0,C 180,E1 11448.707,E2 11448.707} C_VEL
LIN {X 0,Y 232.672,Z 753.746,A -85,B 0,C 180,E1 11443.671,E2 11443.671} C_VEL
LIN {X 0,Y 232.378,Z 757.675,A -85,B 0,C 180,E1 11438.661,E2 11438.661} C_VEL
LIN {X 0,Y 232.486,Z 759.806,A -85,B 0,C 180,E1 11434.192,E2 11434.192} C_VEL
LIN {X 0,Y 232.566,Z 760.618,A -85,B 0,C 180,E1 11430,E2 11430} C_VEL
LIN {X 0,Y 232.44,Z 760.222,A -85,B 0,C 180,E1 11425.559,E2 11425.559} C_VEL
LIN {X 0,Y 232.315,Z 758.574,A -85,B 0,C 180,E1 11421.086,E2 11421.086} C_VEL
LIN {X 0,Y 232.645,Z 755.269,A -85,B 0,C 180,E1 11416.073,E2 11416.073} C_VEL
LIN {X 0,Y 234.06,Z 749.843,A -85,B 0,C 180,E1 11410.536,E2 11410.536} C_VEL
LIN {X 0,Y 236.846,Z 742.711,A -85,B 0,C 180,E1 11405.179,E2 11405.179} C_VEL
LIN {X 0,Y 241.236,Z 733.482,A -85,B 0,C 180,E1 11399.899,E2 11399.899} C_VEL
LIN {X 0,Y 247.148,Z 722.437,A -85,B 0,C 180,E1 11394.937,E2 11394.937} C_VEL
LIN {X 0,Y 253.884,Z 710.456,A -85,B 0,C 180,E1 11390.649,E2 11390.649} C_VEL
LIN {X 0,Y 261.914,Z 696.229,A -85,B 0,C 180,E1 11386.594,E2 11386.594} C_VEL
LIN {X 0,Y 270.628,Z 680.374,A -85,B 0,C 180,E1 11382.985,E2 11382.985} C_VEL
LIN {X 0,Y 279.252,Z 663.879,A -85,B 0,C 180,E1 11379.983,E2 11379.983} C_VEL
LIN {X 0,Y 287.708,Z 646.368,A -85,B 0,C 180,E1 11377.43,E2 11377.43} C_VEL
LIN {X 0,Y 294.297,Z 631.389,A -85,B 0,C 180,E1 11375.637,E2 11375.637} C_VEL
LIN {X 0,Y 287.09,Z 636.015,A -85,B 0,C 180,E1 11374.588,E2 11374.588} C_VEL
LIN {X 0,Y 279.799,Z 640.332,A -85,B 0,C 180,E1 11373.388,E2 11373.388} C_VEL
LIN {X 0,Y 272.291,Z 644.363,A -85,B 0,C 180,E1 11371.922,E2 11371.922} C_VEL
LIN {X 0,Y 265.926,Z 647.367,A -85,B 0,C 180,E1 11370.502,E2 11370.502} C_VEL
LIN {X 0,Y 259.177,Z 658.439,A -85,B 0,C 180,E1 11367.078,E2 11367.078} C_VEL
LIN {X 0,Y 253.982,Z 666.194,A -85,B 0,C 180,E1 11363.921,E2 11363.921} C_VEL
LIN {X 0,Y 249.195,Z 672.521,A -85,B 0,C 180,E1 11360.43,E2 11360.43} C_VEL
LIN {X 0,Y 245.181,Z 676.984,A -85,B 0,C 180,E1 11356.83,E2 11356.83} C_VEL
LIN {X 0,Y 241.907,Z 679.628,A -85,B 0,C 180,E1 11353.139,E2 11353.139} C_VEL
LIN {X 0,Y 239.241,Z 680.631,A -85,B 0,C 180,E1 11349.137,E2 11349.137} C_VEL
LIN {X 0,Y 237.463,Z 679.864,A -85,B 0,C 180,E1 11345.314,E2 11345.314} C_VEL
LIN {X 0,Y 236.253,Z 677.135,A -85,B 0,C 180,E1 11341.212,E2 11341.212} C_VEL
LIN {X 0,Y 235.693,Z 672.831,A -85,B 0,C 180,E1 11337.325,E2 11337.325} C_VEL
LIN {X 0,Y 235.643,Z 666.694,A -85,B 0,C 180,E1 11333.421,E2 11333.421} C_VEL
LIN {X 0,Y 236.12,Z 658.478,A -85,B 0,C 180,E1 11329.508,E2 11329.508} C_VEL
LIN {X 0,Y 237.752,Z 658.567,A -85,B 0,C 180,E1 11327.861,E2 11327.861} C_VEL
LIN {X 0,Y 239.208,Z 658.34,A -85,B 0,C 180,E1 11326.954,E2 11326.954} C_VEL
LIN {X 0,Y 241.563,Z 658.304,A -85,B 0,C 180,E1 11325.374,E2 11325.374} C_VEL
LIN {X 0,Y 245.525,Z 658.049,A -85,B 0,C 180,E1 11323.193,E2 11323.193} C_VEL
LIN {X 0,Y 254.442,Z 657.213,A -85,B 0,C 180,E1 11319.27,E2 11319.27} C_VEL
LIN {X 0,Y 266.363,Z 655.503,A -85,B 0,C 180,E1 11315.375,E2 11315.375} C_VEL
LIN {X 0,Y 276.253,Z 653.685,A -85,B 0,C 180,E1 11312.867,E2 11312.867} C_VEL
LIN {X 0,Y 267.935,Z 667.188,A -85,B 0,C 180,E1 11309.546,E2 11309.546} C_VEL
LIN {X 0,Y 259.94,Z 679.453,A -85,B 0,C 180,E1 11305.792,E2 11305.792} C_VEL
LIN {X 0,Y 252.523,Z 690.417,A -85,B 0,C 180,E1 11301.563,E2 11301.563} C_VEL
LIN {X 0,Y 245.828,Z 700.212,A -85,B 0,C 180,E1 11296.724,E2 11296.724} C_VEL
LIN {X 0,Y 240.522,Z 708.206,A -85,B 0,C 180,E1 11291.558,E2 11291.558} C_VEL
LIN {X 0,Y 236.719,Z 714.334,A -85,B 0,C 180,E1 11286.219,E2 11286.219} C_VEL
LIN {X 0,Y 234.325,Z 718.673,A -85,B 0,C 180,E1 11280.8,E2 11280.8} C_VEL
LIN {X 0,Y 233.144,Z 721.232,A -85,B 0,C 180,E1 11275.668,E2 11275.668} C_VEL
LIN {X 0,Y 232.657,Z 722.394,A -85,B 0,C 180,E1 11270.635,E2 11270.635} C_VEL
LIN {X 0,Y 232.557,Z 722.259,A -85,B 0,C 180,E1 11265.972,E2 11265.972} C_VEL
LIN {X 0,Y 232.689,Z 720.822,A -85,B 0,C 180,E1 11261.15,E2 11261.15} C_VEL
LIN {X 0,Y 233.284,Z 717.967,A -85,B 0,C 180,E1 11256.082,E2 11256.082} C_VEL
LIN {X 0,Y 234.671,Z 713.582,A -85,B 0,C 180,E1 11250.977,E2 11250.977} C_VEL
LIN {X 0,Y 237.242,Z 707.143,A -85,B 0,C 180,E1 11245.65,E2 11245.65} C_VEL
LIN {X 0,Y 240.931,Z 699.209,A -85,B 0,C 180,E1 11240.686,E2 11240.686} C_VEL
LIN {X 0,Y 245.618,Z 689.897,A -85,B 0,C 180,E1 11236.103,E2 11236.103} C_VEL
LIN {X 0,Y 251.123,Z 679.264,A -85,B 0,C 180,E1 11231.907,E2 11231.907} C_VEL
LIN {X 0,Y 257.667,Z 666.626,A -85,B 0,C 180,E1 11227.889,E2 11227.889} C_VEL
LIN {X 0,Y 264.319,Z 653.346,A -85,B 0,C 180,E1 11224.454,E2 11224.454} C_VEL
LIN {X 0,Y 271.25,Z 638.769,A -85,B 0,C 180,E1 11221.367,E2 11221.367} C_VEL
LIN {X 0,Y 278.512,Z 622.15,A -85,B 0,C 180,E1 11218.511,E2 11218.511} C_VEL
LIN {X 0,Y 285.738,Z 603.722,A -85,B 0,C 180,E1 11215.953,E2 11215.953} C_VEL
LIN {X 0,Y 292.242,Z 584.798,A -85,B 0,C 180,E1 11213.843,E2 11213.843} C_VEL
LIN {X 0,Y 298.198,Z 564.386,A -85,B 0,C 180,E1 11212.028,E2 11212.028} C_VEL
LIN {X 0,Y 303.12,Z 543.659,A -85,B 0,C 180,E1 11210.582,E2 11210.582} C_VEL
LIN {X 0,Y 307.007,Z 522.374,A -85,B 0,C 180,E1 11209.448,E2 11209.448} C_VEL
LIN {X 0,Y 311.676,Z 487.28,A -85,B 0,C 180,E1 11208.107,E2 11208.107} C_VEL
LIN {X 0,Y 317.568,Z 444.518,A -85,B 0,C 180,E1 11206.79,E2 11206.79} C_VEL
LIN {X 0,Y 318.018,Z 437.032,A -85,B 0,C 180,E1 11206.426,E2 11206.426} C_VEL
LIN {X 0,Y 317.145,Z 417.475,A -85,B 0,C 180,E1 11204.934,E2 11204.934} C_VEL
LIN {X 0,Y 317.594,Z 411.027,A -85,B 0,C 180,E1 11204.645,E2 11204.645} C_VEL
LIN {X 0,Y 325.116,Z 347.368,A -85,B 0,C 180,E1 11203.053,E2 11203.053} C_VEL
LIN {X 0,Y 325.51,Z 343.057,A -85,B 0,C 180,E1 11202.934,E2 11202.934} C_VEL
LIN {X 0,Y 317.681,Z 333.104,A -85,B 0,C 180,E1 11199.888,E2 11199.888} C_VEL
LIN {X 0,Y 310.896,Z 325.058,A -85,B 0,C 180,E1 11196.914,E2 11196.914} C_VEL
LIN {X 0,Y 305.744,Z 319.596,A -85,B 0,C 180,E1 11194.456,E2 11194.456} C_VEL
LIN {X 0,Y 301.459,Z 315.222,A -85,B 0,C 180,E1 11192.164,E2 11192.164} C_VEL
LIN {X 0,Y 295.784,Z 309.899,A -85,B 0,C 180,E1 11188.687,E2 11188.687} C_VEL
LIN {X 0,Y 287.47,Z 303.39,A -85,B 0,C 180,E1 11181.85,E2 11181.85} C_VEL
LIN {X 0,Y 286.924,Z 303.103,A -85,B 0,C 180,E1 11180.821,E2 11180.821} C_VEL
LIN {X 0,Y 287.114,Z 303.287,A -85,B 0,C 180,E1 11175.555,E2 11175.555} C_VEL
LIN {X 0,Y 288.851,Z 308.006,A -85,B 0,C 180,E1 11167.959,E2 11167.959} C_VEL
LIN {X 0,Y 290.647,Z 312.369,A -85,B 0,C 180,E1 11163.945,E2 11163.945} C_VEL
LIN {X 0,Y 292.587,Z 317.146,A -85,B 0,C 180,E1 11160.588,E2 11160.588} C_VEL
LIN {X 0,Y 295.183,Z 323.533,A -85,B 0,C 180,E1 11156.894,E2 11156.894} C_VEL
LIN {X 0,Y 298.167,Z 331.2,A -85,B 0,C 180,E1 11153.26,E2 11153.26} C_VEL
LIN {X 0,Y 301.414,Z 340.235,A -85,B 0,C 180,E1 11149.682,E2 11149.682} C_VEL
LIN {X 0,Y 305.103,Z 351.308,A -85,B 0,C 180,E1 11145.966,E2 11145.966} C_VEL
LIN {X 0,Y 307.07,Z 357.883,A -85,B 0,C 180,E1 11144.03,E2 11144.03} C_VEL
LIN {X 0,Y 302.721,Z 375.831,A -85,B 0,C 180,E1 11141.925,E2 11141.925} C_VEL
LIN {X 0,Y 305.059,Z 401.878,A -85,B 0,C 180,E1 11139.603,E2 11139.603} C_VEL
LIN {X 0,Y 308.784,Z 427.489,A -85,B 0,C 180,E1 11136.997,E2 11136.997} C_VEL
LIN {X 0,Y 313.521,Z 450.903,A -85,B 0,C 180,E1 11134.271,E2 11134.271} C_VEL
LIN {X 0,Y 318.04,Z 469.287,A -85,B 0,C 180,E1 11131.948,E2 11131.948} C_VEL
LIN {X 0,Y 312.851,Z 494.628,A -85,B 0,C 180,E1 11131.472,E2 11131.472} C_VEL
LIN {X 0,Y 307.31,Z 521.774,A -85,B 0,C 180,E1 11130.506,E2 11130.506} C_VEL
LIN {X 0,Y 299.584,Z 553.222,A -85,B 0,C 180,E1 11129.063,E2 11129.063} C_VEL
LIN {X 0,Y 292.27,Z 579.542,A -85,B 0,C 180,E1 11127.488,E2 11127.488} C_VEL
LIN {X 0,Y 284.162,Z 606.437,A -85,B 0,C 180,E1 11125.422,E2 11125.422} C_VEL
LIN {X 0,Y 277.454,Z 626.539,A -85,B 0,C 180,E1 11123.477,E2 11123.477} C_VEL
LIN {X 0,Y 270.254,Z 645.613,A -85,B 0,C 180,E1 11121.149,E2 11121.149} C_VEL
LIN {X 0,Y 262.777,Z 663.835,A -85,B 0,C 180,E1 11118.389,E2 11118.389} C_VEL
LIN {X 0,Y 255.44,Z 680.347,A -85,B 0,C 180,E1 11115.27,E2 11115.27} C_VEL
LIN {X 0,Y 248.228,Z 695.832,A -85,B 0,C 180,E1 11111.653,E2 11111.653} C_VEL
LIN {X 0,Y 241.803,Z 709.432,A -85,B 0,C 180,E1 11107.733,E2 11107.733} C_VEL
LIN {X 0,Y 235.845,Z 722.13,A -85,B 0,C 180,E1 11103.154,E2 11103.154} C_VEL
LIN {X 0,Y 231.211,Z 732.716,A -85,B 0,C 180,E1 11098.404,E2 11098.404} C_VEL
LIN {X 0,Y 227.854,Z 741.398,A -85,B 0,C 180,E1 11093.493,E2 11093.493} C_VEL
LIN {X 0,Y 225.666,Z 748.48,A -85,B 0,C 180,E1 11088.335,E2 11088.335} C_VEL
LIN {X 0,Y 224.614,Z 753.859,A -85,B 0,C 180,E1 11083.122,E2 11083.122} C_VEL
LIN {X 0,Y 224.402,Z 757.388,A -85,B 0,C 180,E1 11078.197,E2 11078.197} C_VEL
LIN {X 0,Y 224.529,Z 759.341,A -85,B 0,C 180,E1 11073.574,E2 11073.574} C_VEL
LIN {X 0,Y 224.576,Z 759.97,A -85,B 0,C 180,E1 11069.234,E2 11069.234} C_VEL
LIN {X 0,Y 224.437,Z 759.459,A -85,B 0,C 180,E1 11064.888,E2 11064.888} C_VEL
LIN {X 0,Y 224.34,Z 757.558,A -85,B 0,C 180,E1 11059.99,E2 11059.99} C_VEL
LIN {X 0,Y 224.902,Z 753.854,A -85,B 0,C 180,E1 11054.529,E2 11054.529} C_VEL
LIN {X 0,Y 226.624,Z 748.45,A -85,B 0,C 180,E1 11049.061,E2 11049.061} C_VEL
LIN {X 0,Y 229.809,Z 741.242,A -85,B 0,C 180,E1 11043.654,E2 11043.654} C_VEL
LIN {X 0,Y 234.601,Z 732.124,A -85,B 0,C 180,E1 11038.384,E2 11038.384} C_VEL
LIN {X 0,Y 241.075,Z 720.96,A -85,B 0,C 180,E1 11033.327,E2 11033.327} C_VEL
LIN {X 0,Y 248.355,Z 708.844,A -85,B 0,C 180,E1 11028.987,E2 11028.987} C_VEL
LIN {X 0,Y 256.931,Z 694.489,A -85,B 0,C 180,E1 11024.906,E2 11024.906} C_VEL
LIN {X 0,Y 265.705,Z 679.368,A -85,B 0,C 180,E1 11021.474,E2 11021.474} C_VEL
LIN {X 0,Y 274.965,Z 662.342,A -85,B 0,C 180,E1 11018.406,E2 11018.406} C_VEL
LIN {X 0,Y 283.801,Z 644.706,A -85,B 0,C 180,E1 11015.873,E2 11015.873} C_VEL
LIN {X 0,Y 284.965,Z 642.203,A -85,B 0,C 180,E1 11015.56,E2 11015.56} C_VEL
LIN {X 0,Y 277.732,Z 646.224,A -85,B 0,C 180,E1 11014.416,E2 11014.416} C_VEL
LIN {X 0,Y 269.97,Z 650.141,A -85,B 0,C 180,E1 11012.985,E2 11012.985} C_VEL
LIN {X 0,Y 259.818,Z 654.687,A -85,B 0,C 180,E1 11010.785,E2 11010.785} C_VEL
LIN {X 0,Y 257.274,Z 655.622,A -85,B 0,C 180,E1 11010.088,E2 11010.088} C_VEL
LIN {X 0,Y 250.874,Z 664.773,A -85,B 0,C 180,E1 11006.766,E2 11006.766} C_VEL
LIN {X 0,Y 244.929,Z 672.181,A -85,B 0,C 180,E1 11003.072,E2 11003.072} C_VEL
LIN {X 0,Y 240.184,Z 677.257,A -85,B 0,C 180,E1 10999.452,E2 10999.452} C_VEL
LIN {X 0,Y 236.02,Z 680.67,A -85,B 0,C 180,E1 10995.478,E2 10995.478} C_VEL
LIN {X 0,Y 232.755,Z 682.251,A -85,B 0,C 180,E1 10991.396,E2 10991.396} C_VEL
LIN {X 0,Y 230.477,Z 681.99,A -85,B 0,C 180,E1 10987.477,E2 10987.477} C_VEL
LIN {X 0,Y 228.844,Z 679.875,A -85,B 0,C 180,E1 10983.255,E2 10983.255} C_VEL
LIN {X 0,Y 227.971,Z 676.176,A -85,B 0,C 180,E1 10979.245,E2 10979.245} C_VEL
LIN {X 0,Y 227.648,Z 670.658,A -85,B 0,C 180,E1 10975.212,E2 10975.212} C_VEL
LIN {X 0,Y 227.86,Z 663.844,A -85,B 0,C 180,E1 10971.419,E2 10971.419} C_VEL
LIN {X 0,Y 229.354,Z 664.104,A -85,B 0,C 180,E1 10969.703,E2 10969.703} C_VEL
LIN {X 0,Y 230.625,Z 663.948,A -85,B 0,C 180,E1 10968.749,E2 10968.749} C_VEL
LIN {X 0,Y 232.692,Z 663.93,A -85,B 0,C 180,E1 10967.088,E2 10967.088} C_VEL
LIN {X 0,Y 240.194,Z 663.411,A -85,B 0,C 180,E1 10962.559,E2 10962.559} C_VEL
LIN {X 0,Y 249.791,Z 662.45,A -85,B 0,C 180,E1 10958.391,E2 10958.391} C_VEL
LIN {X 0,Y 262.061,Z 660.769,A -85,B 0,C 180,E1 10954.459,E2 10954.459} C_VEL
LIN {X 0,Y 267.764,Z 659.831,A -85,B 0,C 180,E1 10952.958,E2 10952.958} C_VEL
LIN {X 0,Y 258.913,Z 673.171,A -85,B 0,C 180,E1 10949.352,E2 10949.352} C_VEL
LIN {X 0,Y 250.36,Z 685.357,A -85,B 0,C 180,E1 10945.172,E2 10945.172} C_VEL
LIN {X 0,Y 242.556,Z 696.124,A -85,B 0,C 180,E1 10940.431,E2 10940.431} C_VEL
LIN {X 0,Y 236.126,Z 704.992,A -85,B 0,C 180,E1 10935.337,E2 10935.337} C_VEL
LIN {X 0,Y 231.084,Z 712.198,A -85,B 0,C 180,E1 10929.82,E2 10929.82} C_VEL
LIN {X 0,Y 227.689,Z 717.455,A -85,B 0,C 180,E1 10924.201,E2 10924.201} C_VEL
LIN {X 0,Y 225.78,Z 720.841,A -85,B 0,C 180,E1 10918.735,E2 10918.735} C_VEL
LIN {X 0,Y 224.891,Z 722.696,A -85,B 0,C 180,E1 10913.31,E2 10913.31} C_VEL
LIN {X 0,Y 224.598,Z 723.129,A -85,B 0,C 180,E1 10908.158,E2 10908.158} C_VEL
LIN {X 0,Y 224.624,Z 722.296,A -85,B 0,C 180,E1 10903.384,E2 10903.384} C_VEL
LIN {X 0,Y 224.982,Z 720.051,A -85,B 0,C 180,E1 10898.176,E2 10898.176} C_VEL
LIN {X 0,Y 226.085,Z 716.23,A -85,B 0,C 180,E1 10892.789,E2 10892.789} C_VEL
LIN {X 0,Y 228.194,Z 710.844,A -85,B 0,C 180,E1 10887.489,E2 10887.489} C_VEL
LIN {X 0,Y 231.505,Z 703.753,A -85,B 0,C 180,E1 10882.306,E2 10882.306} C_VEL
LIN {X 0,Y 236.116,Z 694.806,A -85,B 0,C 180,E1 10877.28,E2 10877.28} C_VEL
LIN {X 0,Y 241.735,Z 684.406,A -85,B 0,C 180,E1 10872.675,E2 10872.675} C_VEL
LIN {X 0,Y 248.154,Z 672.589,A -85,B 0,C 180,E1 10868.491,E2 10868.491} C_VEL
LIN {X 0,Y 255.168,Z 659.34,A -85,B 0,C 180,E1 10864.716,E2 10864.716} C_VEL
LIN {X 0,Y 262.551,Z 644.63,A -85,B 0,C 180,E1 10861.325,E2 10861.325} C_VEL
LIN {X 0,Y 269.892,Z 628.903,A -85,B 0,C 180,E1 10858.385,E2 10858.385} C_VEL
LIN {X 0,Y 276.718,Z 612.93,A -85,B 0,C 180,E1 10855.941,E2 10855.941} C_VEL
LIN {X 0,Y 283.337,Z 595.598,A -85,B 0,C 180,E1 10853.766,E2 10853.766} C_VEL
LIN {X 0,Y 289.634,Z 576.482,A -85,B 0,C 180,E1 10851.835,E2 10851.835} C_VEL
LIN {X 0,Y 295.219,Z 556.157,A -85,B 0,C 180,E1 10850.2,E2 10850.2} C_VEL
LIN {X 0,Y 299.874,Z 534.937,A -85,B 0,C 180,E1 10848.877,E2 10848.877} C_VEL
LIN {X 0,Y 303.42,Z 513.009,A -85,B 0,C 180,E1 10847.853,E2 10847.853} C_VEL
LIN {X 0,Y 309.62,Z 468.761,A -85,B 0,C 180,E1 10846.309,E2 10846.309} C_VEL
LIN {X 0,Y 317.594,Z 411.027,A -85,B 0,C 180,E1 10844.645,E2 10844.645} C_VEL
LIN {X 0,Y 318.05,Z 403.525,A -85,B 0,C 180,E1 10844.294,E2 10844.294} C_VEL
LIN {X 0,Y 317.261,Z 383.915,A -85,B 0,C 180,E1 10842.824,E2 10842.824} C_VEL
LIN {X 0,Y 317.652,Z 377.448,A -85,B 0,C 180,E1 10842.544,E2 10842.544} C_VEL
LIN {X 0,Y 320.968,Z 347.763,A -85,B 0,C 180,E1 10841.809,E2 10841.809} C_VEL
LIN {X 0,Y 313.089,Z 337.545,A -85,B 0,C 180,E1 10838.517,E2 10838.517} C_VEL
LIN {X 0,Y 305.132,Z 328.367,A -85,B 0,C 180,E1 10834.763,E2 10834.763} C_VEL
LIN {X 0,Y 299.524,Z 322.686,A -85,B 0,C 180,E1 10831.72,E2 10831.72} C_VEL
LIN {X 0,Y 294.048,Z 317.522,A -85,B 0,C 180,E1 10828.275,E2 10828.275} C_VEL
LIN {X 0,Y 286.297,Z 311.279,A -85,B 0,C 180,E1 10821.725,E2 10821.725} C_VEL
LIN {X 0,Y 282.981,Z 310.06,A -85,B 0,C 180,E1 10817.266,E2 10817.266} C_VEL
LIN {X 0,Y 283.191,Z 310.623,A -85,B 0,C 180,E1 10814.937,E2 10814.937} C_VEL
LIN {X 0,Y 284.812,Z 314.894,A -85,B 0,C 180,E1 10808.116,E2 10808.116} C_VEL
LIN {X 0,Y 286.563,Z 319.364,A -85,B 0,C 180,E1 10804.002,E2 10804.002} C_VEL
LIN {X 0,Y 288.346,Z 323.866,A -85,B 0,C 180,E1 10800.795,E2 10800.795} C_VEL
LIN {X 0,Y 290.726,Z 329.938,A -85,B 0,C 180,E1 10797.241,E2 10797.241} C_VEL
LIN {X 0,Y 293.613,Z 337.633,A -85,B 0,C 180,E1 10793.548,E2 10793.548} C_VEL
LIN {X 0,Y 296.735,Z 346.738,A -85,B 0,C 180,E1 10789.909,E2 10789.909} C_VEL
LIN {X 0,Y 300.304,Z 357.935,A -85,B 0,C 180,E1 10786.13,E2 10786.13} C_VEL
LIN {X 0,Y 301.406,Z 362.289,A -85,B 0,C 180,E1 10784.87,E2 10784.87} C_VEL
LIN {X 0,Y 298.948,Z 372.2,A -85,B 0,C 180,E1 10783.729,E2 10783.729} C_VEL
LIN {X 0,Y 300.751,Z 398.77,A -85,B 0,C 180,E1 10781.401,E2 10781.401} C_VEL
LIN {X 0,Y 303.751,Z 423.742,A -85,B 0,C 180,E1 10778.911,E2 10778.911} C_VEL
LIN {X 0,Y 307.683,Z 447.503,A -85,B 0,C 180,E1 10776.187,E2 10776.187} C_VEL
LIN {X 0,Y 312.385,Z 468.557,A -85,B 0,C 180,E1 10773.481,E2 10773.481} C_VEL
LIN {X 0,Y 313.004,Z 471.647,A -85,B 0,C 180,E1 10773.116,E2 10773.116} C_VEL
LIN {X 0,Y 307.715,Z 496.801,A -85,B 0,C 180,E1 10772.609,E2 10772.609} C_VEL
LIN {X 0,Y 301.44,Z 526.079,A -85,B 0,C 180,E1 10771.52,E2 10771.52} C_VEL
LIN {X 0,Y 294.327,Z 553.952,A -85,B 0,C 180,E1 10770.222,E2 10770.222} C_VEL
LIN {X 0,Y 286.506,Z 581.244,A -85,B 0,C 180,E1 10768.568,E2 10768.568} C_VEL
LIN {X 0,Y 278.448,Z 607.317,A -85,B 0,C 180,E1 10766.55,E2 10766.55} C_VEL
LIN {X 0,Y 271.512,Z 627.216,A -85,B 0,C 180,E1 10764.587,E2 10764.587} C_VEL
LIN {X 0,Y 264.204,Z 645.958,A -85,B 0,C 180,E1 10762.273,E2 10762.273} C_VEL
LIN {X 0,Y 256.728,Z 663.394,A -85,B 0,C 180,E1 10759.587,E2 10759.587} C_VEL
LIN {X 0,Y 249.097,Z 679.856,A -85,B 0,C 180,E1 10756.428,E2 10756.428} C_VEL
LIN {X 0,Y 241.571,Z 695.373,A -85,B 0,C 180,E1 10752.749,E2 10752.749} C_VEL
LIN {X 0,Y 234.836,Z 708.933,A -85,B 0,C 180,E1 10748.747,E2 10748.747} C_VEL
LIN {X 0,Y 228.567,Z 721.63,A -85,B 0,C 180,E1 10744.051,E2 10744.051} C_VEL
LIN {X 0,Y 223.667,Z 732.202,A -85,B 0,C 180,E1 10739.16,E2 10739.16} C_VEL
LIN {X 0,Y 219.978,Z 741.176,A -85,B 0,C 180,E1 10733.861,E2 10733.861} C_VEL
LIN {X 0,Y 217.607,Z 748.548,A -85,B 0,C 180,E1 10728.206,E2 10728.206} C_VEL
LIN {X 0,Y 216.588,Z 753.75,A -85,B 0,C 180,E1 10722.802,E2 10722.802} C_VEL
LIN {X 0,Y 216.432,Z 757.079,A -85,B 0,C 180,E1 10717.699,E2 10717.699} C_VEL
LIN {X 0,Y 216.572,Z 758.865,A -85,B 0,C 180,E1 10712.911,E2 10712.911} C_VEL
LIN {X 0,Y 216.592,Z 759.312,A -85,B 0,C 180,E1 10708.677,E2 10708.677} C_VEL
LIN {X 0,Y 216.424,Z 758.687,A -85,B 0,C 180,E1 10704.166,E2 10704.166} C_VEL
LIN {X 0,Y 216.383,Z 756.679,A -85,B 0,C 180,E1 10699.079,E2 10699.079} C_VEL
LIN {X 0,Y 217.132,Z 752.856,A -85,B 0,C 180,E1 10693.411,E2 10693.411} C_VEL
LIN {X 0,Y 219.179,Z 747.343,A -85,B 0,C 180,E1 10687.75,E2 10687.75} C_VEL
LIN {X 0,Y 222.858,Z 739.896,A -85,B 0,C 180,E1 10682.108,E2 10682.108} C_VEL
LIN {X 0,Y 228.429,Z 730.291,A -85,B 0,C 180,E1 10676.528,E2 10676.528} C_VEL
LIN {X 0,Y 235.581,Z 718.902,A -85,B 0,C 180,E1 10671.398,E2 10671.398} C_VEL
LIN {X 0,Y 243.778,Z 706.106,A -85,B 0,C 180,E1 10666.891,E2 10666.891} C_VEL
LIN {X 0,Y 252.715,Z 691.967,A -85,B 0,C 180,E1 10662.949,E2 10662.949} C_VEL
LIN {X 0,Y 262.281,Z 676.098,A -85,B 0,C 180,E1 10659.469,E2 10659.469} C_VEL
LIN {X 0,Y 271.823,Z 659.124,A -85,B 0,C 180,E1 10656.513,E2 10656.513} C_VEL
LIN {X 0,Y 275.443,Z 652.093,A -85,B 0,C 180,E1 10655.442,E2 10655.442} C_VEL
LIN {X 0,Y 264.493,Z 657.274,A -85,B 0,C 180,E1 10653.498,E2 10653.498} C_VEL
LIN {X 0,Y 254.471,Z 661.181,A -85,B 0,C 180,E1 10651.241,E2 10651.241} C_VEL
LIN {X 0,Y 248.58,Z 663.255,A -85,B 0,C 180,E1 10649.652,E2 10649.652} C_VEL
LIN {X 0,Y 242.077,Z 670.95,A -85,B 0,C 180,E1 10646.227,E2 10646.227} C_VEL
LIN {X 0,Y 236.117,Z 677.141,A -85,B 0,C 180,E1 10642.402,E2 10642.402} C_VEL
LIN {X 0,Y 230.835,Z 681.462,A -85,B 0,C 180,E1 10638.171,E2 10638.171} C_VEL
LIN {X 0,Y 226.853,Z 683.66,A -85,B 0,C 180,E1 10634.028,E2 10634.028} C_VEL
LIN {X 0,Y 223.798,Z 683.958,A -85,B 0,C 180,E1 10629.774,E2 10629.774} C_VEL
LIN {X 0,Y 221.662,Z 682.435,A -85,B 0,C 180,E1 10625.435,E2 10625.435} C_VEL
LIN {X 0,Y 220.403,Z 679.293,A -85,B 0,C 180,E1 10621.299,E2 10621.299} C_VEL
LIN {X 0,Y 219.777,Z 674.367,A -85,B 0,C 180,E1 10617.131,E2 10617.131} C_VEL
LIN {X 0,Y 219.728,Z 669.264,A -85,B 0,C 180,E1 10613.729,E2 10613.729} C_VEL
LIN {X 0,Y 221.187,Z 669.39,A -85,B 0,C 180,E1 10611.682,E2 10611.682} C_VEL
LIN {X 0,Y 222.192,Z 669.332,A -85,B 0,C 180,E1 10610.676,E2 10610.676} C_VEL
LIN {X 0,Y 224.397,Z 669.221,A -85,B 0,C 180,E1 10608.693,E2 10608.693} C_VEL
LIN {X 0,Y 227.421,Z 669.11,A -85,B 0,C 180,E1 10606.322,E2 10606.322} C_VEL
LIN {X 0,Y 234.796,Z 668.639,A -85,B 0,C 180,E1 10601.888,E2 10601.888} C_VEL
LIN {X 0,Y 245.117,Z 667.523,A -85,B 0,C 180,E1 10597.452,E2 10597.452} C_VEL
LIN {X 0,Y 257.653,Z 665.815,A -85,B 0,C 180,E1 10593.494,E2 10593.494} C_VEL
LIN {X 0,Y 259.246,Z 665.523,A -85,B 0,C 180,E1 10593.082,E2 10593.082} C_VEL
LIN {X 0,Y 250.093,Z 678.355,A -85,B 0,C 180,E1 10589.268,E2 10589.268} C_VEL
LIN {X 0,Y 241.626,Z 689.618,A -85,B 0,C 180,E1 10585.019,E2 10585.019} C_VEL
LIN {X 0,Y 234.044,Z 699.426,A -85,B 0,C 180,E1 10580.263,E2 10580.263} C_VEL
LIN {X 0,Y 227.627,Z 707.745,A -85,B 0,C 180,E1 10574.991,E2 10574.991} C_VEL
LIN {X 0,Y 222.649,Z 714.404,A -85,B 0,C 180,E1 10569.287,E2 10569.287} C_VEL
LIN {X 0,Y 219.377,Z 719.195,A -85,B 0,C 180,E1 10563.469,E2 10563.469} C_VEL
LIN {X 0,Y 217.632,Z 722.148,A -85,B 0,C 180,E1 10557.945,E2 10557.945} C_VEL
LIN {X 0,Y 216.849,Z 723.612,A -85,B 0,C 180,E1 10552.502,E2 10552.502} C_VEL
LIN {X 0,Y 216.609,Z 723.703,A -85,B 0,C 180,E1 10547.46,E2 10547.46} C_VEL
LIN {X 0,Y 216.67,Z 722.72,A -85,B 0,C 180,E1 10542.527,E2 10542.527} C_VEL
LIN {X 0,Y 217.111,Z 720.368,A -85,B 0,C 180,E1 10537.409,E2 10537.409} C_VEL
LIN {X 0,Y 218.381,Z 716.349,A -85,B 0,C 180,E1 10531.837,E2 10531.837} C_VEL
LIN {X 0,Y 220.771,Z 710.745,A -85,B 0,C 180,E1 10526.365,E2 10526.365} C_VEL
LIN {X 0,Y 224.226,Z 703.86,A -85,B 0,C 180,E1 10521.28,E2 10521.28} C_VEL
LIN {X 0,Y 229.193,Z 694.818,A -85,B 0,C 180,E1 10516.117,E2 10516.117} C_VEL
LIN {X 0,Y 235.192,Z 684.279,A -85,B 0,C 180,E1 10511.407,E2 10511.407} C_VEL
LIN {X 0,Y 242.389,Z 671.606,A -85,B 0,C 180,E1 10506.929,E2 10506.929} C_VEL
LIN {X 0,Y 249.822,Z 658.033,A -85,B 0,C 180,E1 10503.112,E2 10503.112} C_VEL
LIN {X 0,Y 257.132,Z 643.888,A -85,B 0,C 180,E1 10499.893,E2 10499.893} C_VEL
LIN {X 0,Y 264.804,Z 627.878,A -85,B 0,C 180,E1 10496.934,E2 10496.934} C_VEL
LIN {X 0,Y 272.168,Z 610.884,A -85,B 0,C 180,E1 10494.389,E2 10494.389} C_VEL
LIN {X 0,Y 279.425,Z 591.873,A -85,B 0,C 180,E1 10492.096,E2 10492.096} C_VEL
LIN {X 0,Y 285.859,Z 572.145,A -85,B 0,C 180,E1 10490.202,E2 10490.202} C_VEL
LIN {X 0,Y 291.352,Z 551.714,A -85,B 0,C 180,E1 10488.653,E2 10488.653} C_VEL
LIN {X 0,Y 295.785,Z 530.803,A -85,B 0,C 180,E1 10487.43,E2 10487.43} C_VEL
LIN {X 0,Y 299.738,Z 505.353,A -85,B 0,C 180,E1 10486.33,E2 10486.33} C_VEL
LIN {X 0,Y 307.138,Z 455.376,A -85,B 0,C 180,E1 10484.667,E2 10484.667} C_VEL
LIN {X 0,Y 315.981,Z 390.987,A -85,B 0,C 180,E1 10482.884,E2 10482.884} C_VEL
LIN {X 0,Y 317.652,Z 377.448,A -85,B 0,C 180,E1 10482.544,E2 10482.544} C_VEL
LIN {X 0,Y 317.741,Z 372.452,A -85,B 0,C 180,E1 10482.262,E2 10482.262} C_VEL
LIN {X 0,Y 316.163,Z 359.939,A -85,B 0,C 180,E1 10480.98,E2 10480.98} C_VEL
LIN {X 0,Y 316.287,Z 355.624,A -85,B 0,C 180,E1 10480.756,E2 10480.756} C_VEL
LIN {X 0,Y 316.553,Z 352.572,A -85,B 0,C 180,E1 10480.658,E2 10480.658} C_VEL
LIN {X 0,Y 309.564,Z 343.513,A -85,B 0,C 180,E1 10477.564,E2 10477.564} C_VEL
LIN {X 0,Y 302.689,Z 335.45,A -85,B 0,C 180,E1 10474.164,E2 10474.164} C_VEL
LIN {X 0,Y 297.74,Z 330.274,A -85,B 0,C 180,E1 10471.368,E2 10471.368} C_VEL
LIN {X 0,Y 292.433,Z 325.202,A -85,B 0,C 180,E1 10467.932,E2 10467.932} C_VEL
LIN {X 0,Y 285.115,Z 319.17,A -85,B 0,C 180,E1 10461.607,E2 10461.607} C_VEL
LIN {X 0,Y 281.148,Z 317.911,A -85,B 0,C 180,E1 10456.318,E2 10456.318} C_VEL
LIN {X 0,Y 279.488,Z 319.284,A -85,B 0,C 180,E1 10452.186,E2 10452.186} C_VEL
LIN {X 0,Y 280.752,Z 321.646,A -85,B 0,C 180,E1 10448.397,E2 10448.397} C_VEL
LIN {X 0,Y 282.4,Z 326.074,A -85,B 0,C 180,E1 10444.265,E2 10444.265} C_VEL
LIN {X 0,Y 284.109,Z 330.586,A -85,B 0,C 180,E1 10441.009,E2 10441.009} C_VEL
LIN {X 0,Y 286.535,Z 337.127,A -85,B 0,C 180,E1 10437.2,E2 10437.2} C_VEL
LIN {X 0,Y 289.374,Z 344.929,A -85,B 0,C 180,E1 10433.453,E2 10433.453} C_VEL
LIN {X 0,Y 292.579,Z 354.802,A -85,B 0,C 180,E1 10429.566,E2 10429.566} C_VEL
LIN {X 0,Y 295.933,Z 366.124,A -85,B 0,C 180,E1 10425.822,E2 10425.822} C_VEL
LIN {X 0,Y 295.523,Z 368.962,A -85,B 0,C 180,E1 10425.526,E2 10425.526} C_VEL
LIN {X 0,Y 296.764,Z 395.305,A -85,B 0,C 180,E1 10423.258,E2 10423.258} C_VEL
LIN {X 0,Y 299.087,Z 419.91,A -85,B 0,C 180,E1 10420.851,E2 10420.851} C_VEL
LIN {X 0,Y 302.168,Z 443.225,A -85,B 0,C 180,E1 10418.248,E2 10418.248} C_VEL
LIN {X 0,Y 306.503,Z 466.904,A -85,B 0,C 180,E1 10415.243,E2 10415.243} C_VEL
LIN {X 0,Y 308.001,Z 473.915,A -85,B 0,C 180,E1 10414.302,E2 10414.302} C_VEL
LIN {X 0,Y 302.725,Z 498.393,A -85,B 0,C 180,E1 10413.784,E2 10413.784} C_VEL
LIN {X 0,Y 296.065,Z 528.565,A -85,B 0,C 180,E1 10412.646,E2 10412.646} C_VEL
LIN {X 0,Y 287.698,Z 559.855,A -85,B 0,C 180,E1 10411.139,E2 10411.139} C_VEL
LIN {X 0,Y 279.811,Z 586.454,A -85,B 0,C 180,E1 10409.448,E2 10409.448} C_VEL
LIN {X 0,Y 271.377,Z 612.405,A -85,B 0,C 180,E1 10407.339,E2 10407.339} C_VEL
LIN {X 0,Y 264.244,Z 631.605,A -85,B 0,C 180,E1 10405.325,E2 10405.325} C_VEL
LIN {X 0,Y 256.486,Z 650.24,A -85,B 0,C 180,E1 10402.863,E2 10402.863} C_VEL
LIN {X 0,Y 248.619,Z 667.606,A -85,B 0,C 180,E1 10400.007,E2 10400.007} C_VEL
LIN {X 0,Y 240.915,Z 683.337,A -85,B 0,C 180,E1 10396.782,E2 10396.782} C_VEL
LIN {X 0,Y 233.247,Z 698.251,A -85,B 0,C 180,E1 10392.967,E2 10392.967} C_VEL
LIN {X 0,Y 226.073,Z 712.014,A -85,B 0,C 180,E1 10388.579,E2 10388.579} C_VEL
LIN {X 0,Y 219.844,Z 724.088,A -85,B 0,C 180,E1 10383.701,E2 10383.701} C_VEL
LIN {X 0,Y 214.826,Z 734.56,A -85,B 0,C 180,E1 10378.342,E2 10378.342} C_VEL
LIN {X 0,Y 211.353,Z 742.956,A -85,B 0,C 180,E1 10372.825,E2 10372.825} C_VEL
LIN {X 0,Y 209.327,Z 749.447,A -85,B 0,C 180,E1 10367.197,E2 10367.197} C_VEL
LIN {X 0,Y 208.513,Z 754.14,A -85,B 0,C 180,E1 10361.618,E2 10361.618} C_VEL
LIN {X 0,Y 208.492,Z 757.062,A -85,B 0,C 180,E1 10356.332,E2 10356.332} C_VEL
LIN {X 0,Y 208.63,Z 758.4,A -85,B 0,C 180,E1 10351.647,E2 10351.647} C_VEL
LIN {X 0,Y 208.575,Z 758.599,A -85,B 0,C 180,E1 10347.252,E2 10347.252} C_VEL
LIN {X 0,Y 208.385,Z 757.702,A -85,B 0,C 180,E1 10342.556,E2 10342.556} C_VEL
LIN {X 0,Y 208.539,Z 755.193,A -85,B 0,C 180,E1 10336.976,E2 10336.976} C_VEL
LIN {X 0,Y 209.768,Z 750.909,A -85,B 0,C 180,E1 10331.087,E2 10331.087} C_VEL
LIN {X 0,Y 212.67,Z 744.582,A -85,B 0,C 180,E1 10324.967,E2 10324.967} C_VEL
LIN {X 0,Y 217.451,Z 736.323,A -85,B 0,C 180,E1 10319.003,E2 10319.003} C_VEL
LIN {X 0,Y 223.868,Z 726.398,A -85,B 0,C 180,E1 10313.557,E2 10313.557} C_VEL
LIN {X 0,Y 232.063,Z 714.359,A -85,B 0,C 180,E1 10308.431,E2 10308.431} C_VEL
LIN {X 0,Y 240.928,Z 701.326,A -85,B 0,C 180,E1 10304.113,E2 10304.113} C_VEL
LIN {X 0,Y 250.694,Z 686.478,A -85,B 0,C 180,E1 10300.248,E2 10300.248} C_VEL
LIN {X 0,Y 260.781,Z 670.164,A -85,B 0,C 180,E1 10296.926,E2 10296.926} C_VEL
LIN {X 0,Y 266.043,Z 661.073,A -85,B 0,C 180,E1 10295.358,E2 10295.358} C_VEL
LIN {X 0,Y 253.664,Z 665.99,A -85,B 0,C 180,E1 10292.904,E2 10292.904} C_VEL
LIN {X 0,Y 241.638,Z 669.878,A -85,B 0,C 180,E1 10289.771,E2 10289.771} C_VEL
LIN {X 0,Y 239.303,Z 670.519,A -85,B 0,C 180,E1 10288.99,E2 10288.99} C_VEL
LIN {X 0,Y 232.811,Z 676.87,A -85,B 0,C 180,E1 10285.433,E2 10285.433} C_VEL
LIN {X 0,Y 226.875,Z 681.686,A -85,B 0,C 180,E1 10281.455,E2 10281.455} C_VEL
LIN {X 0,Y 221.722,Z 684.794,A -85,B 0,C 180,E1 10277.044,E2 10277.044} C_VEL
LIN {X 0,Y 217.868,Z 685.806,A -85,B 0,C 180,E1 10272.725,E2 10272.725} C_VEL
LIN {X 0,Y 215.025,Z 685.026,A -85,B 0,C 180,E1 10268.287,E2 10268.287} C_VEL
LIN {X 0,Y 213.125,Z 682.412,A -85,B 0,C 180,E1 10263.765,E2 10263.765} C_VEL
LIN {X 0,Y 212.057,Z 677.851,A -85,B 0,C 180,E1 10259.189,E2 10259.189} C_VEL
LIN {X 0,Y 211.804,Z 674.558,A -85,B 0,C 180,E1 10256.481,E2 10256.481} C_VEL
LIN {X 0,Y 213.12,Z 674.613,A -85,B 0,C 180,E1 10254.051,E2 10254.051} C_VEL
LIN {X 0,Y 218.256,Z 674.393,A -85,B 0,C 180,E1 10248.37,E2 10248.37} C_VEL
LIN {X 0,Y 228.316,Z 673.786,A -85,B 0,C 180,E1 10241.62,E2 10241.62} C_VEL
LIN {X 0,Y 242.578,Z 672.259,A -85,B 0,C 180,E1 10235.657,E2 10235.657} C_VEL
LIN {X 0,Y 250.608,Z 671.15,A -85,B 0,C 180,E1 10233.169,E2 10233.169} C_VEL
LIN {X 0,Y 241.141,Z 683.505,A -85,B 0,C 180,E1 10229.127,E2 10229.127} C_VEL
LIN {X 0,Y 232.684,Z 694.009,A -85,B 0,C 180,E1 10224.731,E2 10224.731} C_VEL
LIN {X 0,Y 225.145,Z 703.13,A -85,B 0,C 180,E1 10219.805,E2 10219.805} C_VEL
LIN {X 0,Y 218.846,Z 710.78,A -85,B 0,C 180,E1 10214.349,E2 10214.349} C_VEL
LIN {X 0,Y 214.04,Z 716.851,A -85,B 0,C 180,E1 10208.411,E2 10208.411} C_VEL
LIN {X 0,Y 210.965,Z 721.067,A -85,B 0,C 180,E1 10202.382,E2 10202.382} C_VEL
LIN {X 0,Y 209.409,Z 723.448,A -85,B 0,C 180,E1 10196.668,E2 10196.668} C_VEL
LIN {X 0,Y 208.764,Z 724.43,A -85,B 0,C 180,E1 10191.052,E2 10191.052} C_VEL
LIN {X 0,Y 208.634,Z 724.184,A -85,B 0,C 180,E1 10185.853,E2 10185.853} C_VEL
LIN {X 0,Y 208.792,Z 722.694,A -85,B 0,C 180,E1 10180.764,E2 10180.764} C_VEL
LIN {X 0,Y 209.522,Z 719.793,A -85,B 0,C 180,E1 10175.203,E2 10175.203} C_VEL
LIN {X 0,Y 211.162,Z 715.524,A -85,B 0,C 180,E1 10169.729,E2 10169.729} C_VEL
LIN {X 0,Y 214.266,Z 709.085,A -85,B 0,C 180,E1 10163.839,E2 10163.839} C_VEL
LIN {X 0,Y 218.892,Z 700.71,A -85,B 0,C 180,E1 10158.139,E2 10158.139} C_VEL
LIN {X 0,Y 224.775,Z 690.743,A -85,B 0,C 180,E1 10152.928,E2 10152.928} C_VEL
LIN {X 0,Y 231.669,Z 679.216,A -85,B 0,C 180,E1 10148.213,E2 10148.213} C_VEL
LIN {X 0,Y 239.315,Z 666.136,A -85,B 0,C 180,E1 10143.98,E2 10143.98} C_VEL
LIN {X 0,Y 247.014,Z 652.304,A -85,B 0,C 180,E1 10140.408,E2 10140.408} C_VEL
LIN {X 0,Y 254.908,Z 637.074,A -85,B 0,C 180,E1 10137.228,E2 10137.228} C_VEL
LIN {X 0,Y 262.839,Z 620.313,A -85,B 0,C 180,E1 10134.407,E2 10134.407} C_VEL
LIN {X 0,Y 270.366,Z 602.467,A -85,B 0,C 180,E1 10131.994,E2 10131.994} C_VEL
LIN {X 0,Y 277.01,Z 584.387,A -85,B 0,C 180,E1 10130.023,E2 10130.023} C_VEL
LIN {X 0,Y 283.217,Z 564.426,A -85,B 0,C 180,E1 10128.282,E2 10128.282} C_VEL
LIN {X 0,Y 288.308,Z 544.338,A -85,B 0,C 180,E1 10126.906,E2 10126.906} C_VEL
LIN {X 0,Y 292.362,Z 523.596,A -85,B 0,C 180,E1 10125.814,E2 10125.814} C_VEL
LIN {X 0,Y 298.649,Z 482.406,A -85,B 0,C 180,E1 10124.237,E2 10124.237} C_VEL
LIN {X 0,Y 308.318,Z 418.135,A -85,B 0,C 180,E1 10122.329,E2 10122.329} C_VEL
LIN {X 0,Y 316.225,Z 356.169,A -85,B 0,C 180,E1 10120.769,E2 10120.769} C_VEL
LIN {X 0,Y 316.287,Z 355.624,A -85,B 0,C 180,E1 10120.756,E2 10120.756} C_VEL
LIN {X 0,Y 316.049,Z 353.486,A -85,B 0,C 180,E1 10120.543,E2 10120.543} C_VEL
LIN {X 0,Y 314.922,Z 351.863,A -85,B 0,C 180,E1 10120.055,E2 10120.055} C_VEL
LIN {X 0,Y 312.705,Z 351.108,A -85,B 0,C 180,E1 10119.224,E2 10119.224} C_VEL
LIN {X 0,Y 308.299,Z 351.166,A -85,B 0,C 180,E1 10117.58,E2 10117.58} C_VEL
LIN {X 0,Y 306.606,Z 350.078,A -85,B 0,C 180,E1 10116.846,E2 10116.846} C_VEL
LIN {X 0,Y 300.259,Z 342.515,A -85,B 0,C 180,E1 10113.559,E2 10113.559} C_VEL
LIN {X 0,Y 295.808,Z 337.728,A -85,B 0,C 180,E1 10110.916,E2 10110.916} C_VEL
LIN {X 0,Y 290.905,Z 332.932,A -85,B 0,C 180,E1 10107.647,E2 10107.647} C_VEL
LIN {X 0,Y 283.744,Z 326.963,A -85,B 0,C 180,E1 10101.282,E2 10101.282} C_VEL
LIN {X 0,Y 280.031,Z 325.84,A -85,B 0,C 180,E1 10096.164,E2 10096.164} C_VEL
LIN {X 0,Y 277.765,Z 328.703,A -85,B 0,C 180,E1 10088.905,E2 10088.905} C_VEL
LIN {X 0,Y 278.167,Z 332.497,A -85,B 0,C 180,E1 10084.743,E2 10084.743} C_VEL
LIN {X 0,Y 279.877,Z 337.304,A -85,B 0,C 180,E1 10081.229,E2 10081.229} C_VEL
LIN {X 0,Y 282.281,Z 344.098,A -85,B 0,C 180,E1 10077.264,E2 10077.264} C_VEL
LIN {X 0,Y 284.95,Z 351.82,A -85,B 0,C 180,E1 10073.554,E2 10073.554} C_VEL
LIN {X 0,Y 287.499,Z 359.094,A -85,B 0,C 180,E1 10070.745,E2 10070.745} C_VEL
LIN {X 0,Y 292.485,Z 371.442,A -85,B 0,C 180,E1 10066.886,E2 10066.886} C_VEL
LIN {X 0,Y 293.488,Z 398.325,A -85,B 0,C 180,E1 10064.552,E2 10064.552} C_VEL
LIN {X 0,Y 295.47,Z 423.405,A -85,B 0,C 180,E1 10062.053,E2 10062.053} C_VEL
LIN {X 0,Y 298.314,Z 447.692,A -85,B 0,C 180,E1 10059.282,E2 10059.282} C_VEL
LIN {X 0,Y 302.198,Z 471.524,A -85,B 0,C 180,E1 10056.168,E2 10056.168} C_VEL
LIN {X 0,Y 303.079,Z 476.48,A -85,B 0,C 180,E1 10055.52,E2 10055.52} C_VEL
LIN {X 0,Y 297.928,Z 499.829,A -85,B 0,C 180,E1 10055.005,E2 10055.005} C_VEL
LIN {X 0,Y 291.197,Z 529.201,A -85,B 0,C 180,E1 10053.882,E2 10053.882} C_VEL
LIN {X 0,Y 283.046,Z 559.199,A -85,B 0,C 180,E1 10052.456,E2 10052.456} C_VEL
LIN {X 0,Y 274.486,Z 587.203,A -85,B 0,C 180,E1 10050.675,E2 10050.675} C_VEL
LIN {X 0,Y 266.622,Z 611.003,A -85,B 0,C 180,E1 10048.762,E2 10048.762} C_VEL
LIN {X 0,Y 259.348,Z 630.124,A -85,B 0,C 180,E1 10046.782,E2 10046.782} C_VEL
LIN {X 0,Y 251.2,Z 649.156,A -85,B 0,C 180,E1 10044.29,E2 10044.29} C_VEL
LIN {X 0,Y 243.011,Z 666.581,A -85,B 0,C 180,E1 10041.421,E2 10041.421} C_VEL
LIN {X 0,Y 234.593,Z 683.04,A -85,B 0,C 180,E1 10038,E2 10038} C_VEL
LIN {X 0,Y 226.699,Z 697.758,A -85,B 0,C 180,E1 10034.175,E2 10034.175} C_VEL
LIN {X 0,Y 219.559,Z 710.804,A -85,B 0,C 180,E1 10029.949,E2 10029.949} C_VEL
LIN {X 0,Y 213.23,Z 722.398,A -85,B 0,C 180,E1 10025.223,E2 10025.223} C_VEL
LIN {X 0,Y 207.979,Z 732.559,A -85,B 0,C 180,E1 10019.998,E2 10019.998} C_VEL
LIN {X 0,Y 204.044,Z 741.262,A -85,B 0,C 180,E1 10014.297,E2 10014.297} C_VEL
LIN {X 0,Y 201.653,Z 748.011,A -85,B 0,C 180,E1 10008.501,E2 10008.501} C_VEL
LIN {X 0,Y 200.6,Z 752.95,A -85,B 0,C 180,E1 10002.668,E2 10002.668} C_VEL
LIN {X 0,Y 200.494,Z 756.119,A -85,B 0,C 180,E1 9997.071,E2 9997.071} C_VEL
LIN {X 0,Y 200.646,Z 757.62,A -85,B 0,C 180,E1 9992.284,E2 9992.284} C_VEL
LIN {X 0,Y 200.616,Z 757.983,A -85,B 0,C 180,E1 9987.714,E2 9987.714} C_VEL
LIN {X 0,Y 200.413,Z 757.21,A -85,B 0,C 180,E1 9982.835,E2 9982.835} C_VEL
LIN {X 0,Y 200.538,Z 754.906,A -85,B 0,C 180,E1 9977.034,E2 9977.034} C_VEL
LIN {X 0,Y 201.793,Z 750.864,A -85,B 0,C 180,E1 9970.911,E2 9970.911} C_VEL
LIN {X 0,Y 204.812,Z 744.768,A -85,B 0,C 180,E1 9964.557,E2 9964.557} C_VEL
LIN {X 0,Y 209.802,Z 736.714,A -85,B 0,C 180,E1 9958.383,E2 9958.383} C_VEL
LIN {X 0,Y 216.497,Z 727.125,A -85,B 0,C 180,E1 9952.77,E2 9952.77} C_VEL
LIN {X 0,Y 224.575,Z 716.003,A -85,B 0,C 180,E1 9947.756,E2 9947.756} C_VEL
LIN {X 0,Y 233.69,Z 703.397,A -85,B 0,C 180,E1 9943.334,E2 9943.334} C_VEL
LIN {X 0,Y 244.086,Z 688.49,A -85,B 0,C 180,E1 9939.266,E2 9939.266} C_VEL
LIN {X 0,Y 254.385,Z 672.913,A -85,B 0,C 180,E1 9935.934,E2 9935.934} C_VEL
LIN {X 0,Y 256.498,Z 669.332,A -85,B 0,C 180,E1 9935.233,E2 9935.233} C_VEL
LIN {X 0,Y 243.197,Z 673.75,A -85,B 0,C 180,E1 9932.307,E2 9932.307} C_VEL
LIN {X 0,Y 231.106,Z 676.929,A -85,B 0,C 180,E1 9928.7,E2 9928.7} C_VEL
LIN {X 0,Y 229.046,Z 677.634,A -85,B 0,C 180,E1 9927.845,E2 9927.845} C_VEL
LIN {X 0,Y 222.32,Z 682.746,A -85,B 0,C 180,E1 9923.875,E2 9923.875} C_VEL
LIN {X 0,Y 216.652,Z 686.01,A -85,B 0,C 180,E1 9919.687,E2 9919.687} C_VEL
LIN {X 0,Y 211.822,Z 687.527,A -85,B 0,C 180,E1 9915.046,E2 9915.046} C_VEL
LIN {X 0,Y 208.36,Z 687.151,A -85,B 0,C 180,E1 9910.506,E2 9910.506} C_VEL
LIN {X 0,Y 205.929,Z 684.906,A -85,B 0,C 180,E1 9905.851,E2 9905.851} C_VEL
LIN {X 0,Y 204.455,Z 680.849,A -85,B 0,C 180,E1 9901.12,E2 9901.12} C_VEL
LIN {X 0,Y 204.247,Z 679.746,A -85,B 0,C 180,E1 9899.999,E2 9899.999} C_VEL
LIN {X 0,Y 205.221,Z 679.71,A -85,B 0,C 180,E1 9896.927,E2 9896.927} C_VEL
LIN {X 0,Y 209.687,Z 679.407,A -85,B 0,C 180,E1 9890.392,E2 9890.392} C_VEL
LIN {X 0,Y 215.583,Z 679.108,A -85,B 0,C 180,E1 9885.22,E2 9885.22} C_VEL
LIN {X 0,Y 226.881,Z 678.217,A -85,B 0,C 180,E1 9878.815,E2 9878.815} C_VEL
LIN {X 0,Y 241.194,Z 676.525,A -85,B 0,C 180,E1 9873.563,E2 9873.563} C_VEL
LIN {X 0,Y 242.017,Z 676.446,A -85,B 0,C 180,E1 9873.295,E2 9873.295} C_VEL
LIN {X 0,Y 232.169,Z 688.417,A -85,B 0,C 180,E1 9868.984,E2 9868.984} C_VEL
LIN {X 0,Y 223.072,Z 698.907,A -85,B 0,C 180,E1 9864.042,E2 9864.042} C_VEL
LIN {X 0,Y 215.148,Z 707.834,A -85,B 0,C 180,E1 9858.437,E2 9858.437} C_VEL
LIN {X 0,Y 209.102,Z 714.71,A -85,B 0,C 180,E1 9852.575,E2 9852.575} C_VEL
LIN {X 0,Y 204.72,Z 719.942,A -85,B 0,C 180,E1 9846.226,E2 9846.226} C_VEL
LIN {X 0,Y 202.198,Z 723.24,A -85,B 0,C 180,E1 9839.964,E2 9839.964} C_VEL
LIN {X 0,Y 201.056,Z 724.83,A -85,B 0,C 180,E1 9834.067,E2 9834.067} C_VEL
LIN {X 0,Y 200.678,Z 725.071,A -85,B 0,C 180,E1 9828.294,E2 9828.294} C_VEL
LIN {X 0,Y 200.711,Z 724.147,A -85,B 0,C 180,E1 9822.955,E2 9822.955} C_VEL
LIN {X 0,Y 201.157,Z 721.87,A -85,B 0,C 180,E1 9817.426,E2 9817.426} C_VEL
LIN {X 0,Y 202.536,Z 717.944,A -85,B 0,C 180,E1 9811.415,E2 9811.415} C_VEL
LIN {X 0,Y 205.165,Z 712.431,A -85,B 0,C 180,E1 9805.528,E2 9805.528} C_VEL
LIN {X 0,Y 209.199,Z 705.224,A -85,B 0,C 180,E1 9799.815,E2 9799.815} C_VEL
LIN {X 0,Y 214.729,Z 696.168,A -85,B 0,C 180,E1 9794.332,E2 9794.332} C_VEL
LIN {X 0,Y 221.352,Z 685.635,A -85,B 0,C 180,E1 9789.37,E2 9789.37} C_VEL
LIN {X 0,Y 228.817,Z 673.616,A -85,B 0,C 180,E1 9784.922,E2 9784.922} C_VEL
LIN {X 0,Y 236.855,Z 660.133,A -85,B 0,C 180,E1 9780.958,E2 9780.958} C_VEL
LIN {X 0,Y 245.238,Z 645.147,A -85,B 0,C 180,E1 9777.441,E2 9777.441} C_VEL
LIN {X 0,Y 253.489,Z 629.056,A -85,B 0,C 180,E1 9774.423,E2 9774.423} C_VEL
LIN {X 0,Y 261.367,Z 611.952,A -85,B 0,C 180,E1 9771.843,E2 9771.843} C_VEL
LIN {X 0,Y 268.698,Z 593.878,A -85,B 0,C 180,E1 9769.649,E2 9769.649} C_VEL
LIN {X 0,Y 275.342,Z 574.809,A -85,B 0,C 180,E1 9767.794,E2 9767.794} C_VEL
LIN {X 0,Y 281.167,Z 554.628,A -85,B 0,C 180,E1 9766.238,E2 9766.238} C_VEL
LIN {X 0,Y 286.022,Z 533.32,A -85,B 0,C 180,E1 9764.972,E2 9764.972} C_VEL
LIN {X 0,Y 290.521,Z 506.454,A -85,B 0,C 180,E1 9763.8,E2 9763.8} C_VEL
LIN {X 0,Y 298.037,Z 459.915,A -85,B 0,C 180,E1 9762.22,E2 9762.22} C_VEL
LIN {X 0,Y 307.406,Z 396.463,A -85,B 0,C 180,E1 9760.457,E2 9760.457} C_VEL
LIN {X 0,Y 312.255,Z 357.41,A -85,B 0,C 180,E1 9759.478,E2 9759.478} C_VEL
LIN {X 0,Y 306.606,Z 350.078,A -85,B 0,C 180,E1 9756.846,E2 9756.846} C_VEL
LIN {X 0,Y 303.833,Z 347.906,A -85,B 0,C 180,E1 9755.55,E2 9755.55} C_VEL
LIN {X 0,Y 298.815,Z 346.893,A -85,B 0,C 180,E1 9753.188,E2 9753.188} C_VEL
LIN {X 0,Y 294.784,Z 345.882,A -85,B 0,C 180,E1 9751.049,E2 9751.049} C_VEL
LIN {X 0,Y 293.94,Z 345.274,A -85,B 0,C 180,E1 9750.541,E2 9750.541} C_VEL
LIN {X 0,Y 289.358,Z 340.658,A -85,B 0,C 180,E1 9747.36,E2 9747.36} C_VEL
LIN {X 0,Y 282.566,Z 334.855,A -85,B 0,C 180,E1 9741.158,E2 9741.158} C_VEL
LIN {X 0,Y 278.917,Z 333.766,A -85,B 0,C 180,E1 9736.024,E2 9736.024} C_VEL
LIN {X 0,Y 276.715,Z 336.773,A -85,B 0,C 180,E1 9728.939,E2 9728.939} C_VEL
LIN {X 0,Y 276.921,Z 340.384,A -85,B 0,C 180,E1 9724.972,E2 9724.972} C_VEL
LIN {X 0,Y 278.171,Z 345.672,A -85,B 0,C 180,E1 9721.03,E2 9721.03} C_VEL
LIN {X 0,Y 280.734,Z 353.399,A -85,B 0,C 180,E1 9716.683,E2 9716.683} C_VEL
LIN {X 0,Y 284.249,Z 362.608,A -85,B 0,C 180,E1 9712.675,E2 9712.675} C_VEL
LIN {X 0,Y 288.727,Z 374.369,A -85,B 0,C 180,E1 9708.717,E2 9708.717} C_VEL
LIN {X 0,Y 289.59,Z 376.937,A -85,B 0,C 180,E1 9708.032,E2 9708.032} C_VEL
LIN {X 0,Y 290.544,Z 405.409,A -85,B 0,C 180,E1 9705.489,E2 9705.489} C_VEL
LIN {X 0,Y 292.366,Z 432.148,A -85,B 0,C 180,E1 9702.704,E2 9702.704} C_VEL
LIN {X 0,Y 294.929,Z 456.106,A -85,B 0,C 180,E1 9699.822,E2 9699.822} C_VEL
LIN {X 0,Y 298.296,Z 478.903,A -85,B 0,C 180,E1 9696.775,E2 9696.775} C_VEL
LIN {X 0,Y 293.113,Z 501.873,A -85,B 0,C 180,E1 9696.241,E2 9696.241} C_VEL
LIN {X 0,Y 285.269,Z 534.683,A -85,B 0,C 180,E1 9694.962,E2 9694.962} C_VEL
LIN {X 0,Y 276.433,Z 565.44,A -85,B 0,C 180,E1 9693.419,E2 9693.419} C_VEL
LIN {X 0,Y 268.331,Z 591.155,A -85,B 0,C 180,E1 9691.729,E2 9691.729} C_VEL
LIN {X 0,Y 260.986,Z 612.285,A -85,B 0,C 180,E1 9689.977,E2 9689.977} C_VEL
LIN {X 0,Y 253.515,Z 631.13,A -85,B 0,C 180,E1 9687.99,E2 9687.99} C_VEL
LIN {X 0,Y 245.446,Z 649.348,A -85,B 0,C 180,E1 9685.579,E2 9685.579} C_VEL
LIN {X 0,Y 236.971,Z 666.635,A -85,B 0,C 180,E1 9682.687,E2 9682.687} C_VEL
LIN {X 0,Y 228.316,Z 682.905,A -85,B 0,C 180,E1 9679.254,E2 9679.254} C_VEL
LIN {X 0,Y 219.789,Z 698.109,A -85,B 0,C 180,E1 9675.208,E2 9675.208} C_VEL
LIN {X 0,Y 212.359,Z 710.957,A -85,B 0,C 180,E1 9670.878,E2 9670.878} C_VEL
LIN {X 0,Y 205.434,Z 723.009,A -85,B 0,C 180,E1 9665.735,E2 9665.735} C_VEL
LIN {X 0,Y 200.032,Z 732.991,A -85,B 0,C 180,E1 9660.321,E2 9660.321} C_VEL
LIN {X 0,Y 196.007,Z 741.441,A -85,B 0,C 180,E1 9654.405,E2 9654.405} C_VEL
LIN {X 0,Y 193.595,Z 747.967,A -85,B 0,C 180,E1 9648.363,E2 9648.363} C_VEL
LIN {X 0,Y 192.584,Z 752.74,A -85,B 0,C 180,E1 9642.29,E2 9642.29} C_VEL
LIN {X 0,Y 192.536,Z 755.7,A -85,B 0,C 180,E1 9636.56,E2 9636.56} C_VEL
LIN {X 0,Y 192.69,Z 757.061,A -85,B 0,C 180,E1 9631.486,E2 9631.486} C_VEL
LIN {X 0,Y 192.602,Z 757.27,A -85,B 0,C 180,E1 9626.726,E2 9626.726} C_VEL
LIN {X 0,Y 192.392,Z 756.358,A -85,B 0,C 180,E1 9621.632,E2 9621.632} C_VEL
LIN {X 0,Y 192.709,Z 753.868,A -85,B 0,C 180,E1 9615.578,E2 9615.578} C_VEL
LIN {X 0,Y 194.356,Z 749.605,A -85,B 0,C 180,E1 9609.208,E2 9609.208} C_VEL
LIN {X 0,Y 197.964,Z 743.306,A -85,B 0,C 180,E1 9602.637,E2 9602.637} C_VEL
LIN {X 0,Y 203.678,Z 735.1,A -85,B 0,C 180,E1 9596.308,E2 9596.308} C_VEL
LIN {X 0,Y 211.356,Z 724.978,A -85,B 0,C 180,E1 9590.451,E2 9590.451} C_VEL
LIN {X 0,Y 220.404,Z 713.283,A -85,B 0,C 180,E1 9585.319,E2 9585.319} C_VEL
LIN {X 0,Y 230.839,Z 699.621,A -85,B 0,C 180,E1 9580.711,E2 9580.711} C_VEL
LIN {X 0,Y 241.599,Z 684.879,A -85,B 0,C 180,E1 9576.875,E2 9576.875} C_VEL
LIN {X 0,Y 247.134,Z 676.845,A -85,B 0,C 180,E1 9575.142,E2 9575.142} C_VEL
LIN {X 0,Y 234.021,Z 680.516,A -85,B 0,C 180,E1 9571.991,E2 9571.991} C_VEL
LIN {X 0,Y 221.826,Z 683.163,A -85,B 0,C 180,E1 9567.954,E2 9567.954} C_VEL
LIN {X 0,Y 218.272,Z 683.85,A -85,B 0,C 180,E1 9566.38,E2 9566.38} C_VEL
LIN {X 0,Y 211.455,Z 687.545,A -85,B 0,C 180,E1 9561.934,E2 9561.934} C_VEL
LIN {X 0,Y 206.173,Z 689.224,A -85,B 0,C 180,E1 9557.497,E2 9557.497} C_VEL
LIN {X 0,Y 201.802,Z 689.104,A -85,B 0,C 180,E1 9552.591,E2 9552.591} C_VEL
LIN {X 0,Y 198.845,Z 687.194,A -85,B 0,C 180,E1 9547.802,E2 9547.802} C_VEL
LIN {X 0,Y 197.423,Z 684.919,A -85,B 0,C 180,E1 9544.356,E2 9544.356} C_VEL
LIN {X 0,Y 197.759,Z 684.693,A -85,B 0,C 180,E1 9540.289,E2 9540.289} C_VEL
LIN {X 0,Y 199.001,Z 684.554,A -85,B 0,C 180,E1 9536.542,E2 9536.542} C_VEL
LIN {X 0,Y 206.352,Z 684.035,A -85,B 0,C 180,E1 9527.12,E2 9527.12} C_VEL
LIN {X 0,Y 217.424,Z 683.202,A -85,B 0,C 180,E1 9519.823,E2 9519.823} C_VEL
LIN {X 0,Y 231.828,Z 681.649,A -85,B 0,C 180,E1 9513.9,E2 9513.9} C_VEL
LIN {X 0,Y 233.197,Z 681.605,A -85,B 0,C 180,E1 9513.366,E2 9513.366} C_VEL
LIN {X 0,Y 223.167,Z 692.958,A -85,B 0,C 180,E1 9508.843,E2 9508.843} C_VEL
LIN {X 0,Y 214.27,Z 702.515,A -85,B 0,C 180,E1 9503.832,E2 9503.832} C_VEL
LIN {X 0,Y 206.592,Z 710.564,A -85,B 0,C 180,E1 9498.188,E2 9498.188} C_VEL
LIN {X 0,Y 200.532,Z 716.967,A -85,B 0,C 180,E1 9492.018,E2 9492.018} C_VEL
LIN {X 0,Y 196.322,Z 721.628,A -85,B 0,C 180,E1 9485.493,E2 9485.493} C_VEL
LIN {X 0,Y 193.906,Z 724.552,A -85,B 0,C 180,E1 9478.764,E2 9478.764} C_VEL
LIN {X 0,Y 192.956,Z 725.74,A -85,B 0,C 180,E1 9472.724,E2 9472.724} C_VEL
LIN {X 0,Y 192.684,Z 725.614,A -85,B 0,C 180,E1 9467.205,E2 9467.205} C_VEL
LIN {X 0,Y 192.784,Z 724.359,A -85,B 0,C 180,E1 9461.67,E2 9461.67} C_VEL
LIN {X 0,Y 193.424,Z 721.887,A -85,B 0,C 180,E1 9455.935,E2 9455.935} C_VEL
LIN {X 0,Y 195.156,Z 717.602,A -85,B 0,C 180,E1 9449.707,E2 9449.707} C_VEL
LIN {X 0,Y 198.243,Z 711.71,A -85,B 0,C 180,E1 9443.63,E2 9443.63} C_VEL
LIN {X 0,Y 202.864,Z 704.093,A -85,B 0,C 180,E1 9437.765,E2 9437.765} C_VEL
LIN {X 0,Y 209.031,Z 694.594,A -85,B 0,C 180,E1 9432.174,E2 9432.174} C_VEL
LIN {X 0,Y 216.282,Z 683.574,A -85,B 0,C 180,E1 9427.15,E2 9427.15} C_VEL
LIN {X 0,Y 224.366,Z 671.037,A -85,B 0,C 180,E1 9422.677,E2 9422.677} C_VEL
LIN {X 0,Y 232.982,Z 656.964,A -85,B 0,C 180,E1 9418.716,E2 9418.716} C_VEL
LIN {X 0,Y 241.618,Z 641.769,A -85,B 0,C 180,E1 9415.32,E2 9415.32} C_VEL
LIN {X 0,Y 250.298,Z 624.96,A -85,B 0,C 180,E1 9412.325,E2 9412.325} C_VEL
LIN {X 0,Y 258.564,Z 606.982,A -85,B 0,C 180,E1 9409.776,E2 9409.776} C_VEL
LIN {X 0,Y 266.217,Z 587.778,A -85,B 0,C 180,E1 9407.611,E2 9407.611} C_VEL
LIN {X 0,Y 272.798,Z 568.197,A -85,B 0,C 180,E1 9405.862,E2 9405.862} C_VEL
LIN {X 0,Y 278.185,Z 548.627,A -85,B 0,C 180,E1 9404.484,E2 9404.484} C_VEL
LIN {X 0,Y 282.755,Z 527.266,A -85,B 0,C 180,E1 9403.327,E2 9403.327} C_VEL
LIN {X 0,Y 289.536,Z 486.766,A -85,B 0,C 180,E1 9401.725,E2 9401.725} C_VEL
LIN {X 0,Y 299.652,Z 424.381,A -85,B 0,C 180,E1 9399.856,E2 9399.856} C_VEL
LIN {X 0,Y 307.744,Z 365.74,A -85,B 0,C 180,E1 9398.376,E2 9398.376} C_VEL
LIN {X 0,Y 308.137,Z 362.474,A -85,B 0,C 180,E1 9398.3,E2 9398.3} C_VEL
LIN {X 0,Y 301.895,Z 354.351,A -85,B 0,C 180,E1 9395.19,E2 9395.19} C_VEL
LIN {X 0,Y 296.269,Z 347.733,A -85,B 0,C 180,E1 9391.996,E2 9391.996} C_VEL
LIN {X 0,Y 293.94,Z 345.274,A -85,B 0,C 180,E1 9390.541,E2 9390.541} C_VEL
LIN {X 0,Y 291.59,Z 344.32,A -85,B 0,C 180,E1 9389.102,E2 9389.102} C_VEL
LIN {X 0,Y 285.187,Z 345.758,A -85,B 0,C 180,E1 9384.832,E2 9384.832} C_VEL
LIN {X 0,Y 283.93,Z 345.156,A -85,B 0,C 180,E1 9383.741,E2 9383.741} C_VEL
LIN {X 0,Y 281.203,Z 342.69,A -85,B 0,C 180,E1 9380.829,E2 9380.829} C_VEL
LIN {X 0,Y 277.904,Z 341.7,A -85,B 0,C 180,E1 9376.084,E2 9376.084} C_VEL
LIN {X 0,Y 275.688,Z 344.632,A -85,B 0,C 180,E1 9369.183,E2 9369.183} C_VEL
LIN {X 0,Y 275.796,Z 348.153,A -85,B 0,C 180,E1 9365.305,E2 9365.305} C_VEL
LIN {X 0,Y 276.965,Z 353.455,A -85,B 0,C 180,E1 9361.345,E2 9361.345} C_VEL
LIN {X 0,Y 279.375,Z 361.289,A -85,B 0,C 180,E1 9356.989,E2 9356.989} C_VEL
LIN {X 0,Y 282.613,Z 370.189,A -85,B 0,C 180,E1 9353.143,E2 9353.143} C_VEL
LIN {X 0,Y 286.809,Z 381.83,A -85,B 0,C 180,E1 9349.239,E2 9349.239} C_VEL
LIN {X 0,Y 287.546,Z 410.565,A -85,B 0,C 180,E1 9346.618,E2 9346.618} C_VEL
LIN {X 0,Y 288.906,Z 436.991,A -85,B 0,C 180,E1 9343.785,E2 9343.785} C_VEL
LIN {X 0,Y 291.104,Z 461.249,A -85,B 0,C 180,E1 9340.781,E2 9340.781} C_VEL
LIN {X 0,Y 293.688,Z 481.107,A -85,B 0,C 180,E1 9338.072,E2 9338.072} C_VEL
LIN {X 0,Y 288.239,Z 504.765,A -85,B 0,C 180,E1 9337.487,E2 9337.487} C_VEL
LIN {X 0,Y 280.868,Z 534.54,A -85,B 0,C 180,E1 9336.316,E2 9336.316} C_VEL
LIN {X 0,Y 272.048,Z 564.858,A -85,B 0,C 180,E1 9334.829,E2 9334.829} C_VEL
LIN {X 0,Y 263.472,Z 591.267,A -85,B 0,C 180,E1 9333.101,E2 9333.101} C_VEL
LIN {X 0,Y 256.669,Z 610.502,A -85,B 0,C 180,E1 9331.534,E2 9331.534} C_VEL
LIN {X 0,Y 249.177,Z 629.036,A -85,B 0,C 180,E1 9329.623,E2 9329.623} C_VEL
LIN {X 0,Y 241.124,Z 646.777,A -85,B 0,C 180,E1 9327.327,E2 9327.327} C_VEL
LIN {X 0,Y 232.382,Z 664.186,A -85,B 0,C 180,E1 9324.49,E2 9324.49} C_VEL
LIN {X 0,Y 223.467,Z 680.405,A -85,B 0,C 180,E1 9321.126,E2 9321.126} C_VEL
LIN {X 0,Y 214.599,Z 695.619,A -85,B 0,C 180,E1 9317.139,E2 9317.139} C_VEL
LIN {X 0,Y 206.497,Z 709.043,A -85,B 0,C 180,E1 9312.678,E2 9312.678} C_VEL
LIN {X 0,Y 199.095,Z 721.173,A -85,B 0,C 180,E1 9307.49,E2 9307.49} C_VEL
LIN {X 0,Y 193.123,Z 731.446,A -85,B 0,C 180,E1 9301.876,E2 9301.876} C_VEL
LIN {X 0,Y 188.609,Z 740.217,A -85,B 0,C 180,E1 9295.685,E2 9295.685} C_VEL
LIN {X 0,Y 185.8,Z 747.099,A -85,B 0,C 180,E1 9289.163,E2 9289.163} C_VEL
LIN {X 0,Y 184.637,Z 751.936,A -85,B 0,C 180,E1 9282.828,E2 9282.828} C_VEL
LIN {X 0,Y 184.548,Z 754.955,A -85,B 0,C 180,E1 9276.845,E2 9276.845} C_VEL
LIN {X 0,Y 184.711,Z 756.324,A -85,B 0,C 180,E1 9271.861,E2 9271.861} C_VEL
LIN {X 0,Y 184.648,Z 756.642,A -85,B 0,C 180,E1 9267.206,E2 9267.206} C_VEL
LIN {X 0,Y 184.418,Z 755.872,A -85,B 0,C 180,E1 9261.896,E2 9261.896} C_VEL
LIN {X 0,Y 184.709,Z 753.572,A -85,B 0,C 180,E1 9255.581,E2 9255.581} C_VEL
LIN {X 0,Y 186.407,Z 749.54,A -85,B 0,C 180,E1 9248.937,E2 9248.937} C_VEL
LIN {X 0,Y 190.177,Z 743.523,A -85,B 0,C 180,E1 9242.1,E2 9242.1} C_VEL
LIN {X 0,Y 196.152,Z 735.538,A -85,B 0,C 180,E1 9235.541,E2 9235.541} C_VEL
LIN {X 0,Y 203.913,Z 725.963,A -85,B 0,C 180,E1 9229.665,E2 9229.665} C_VEL
LIN {X 0,Y 213.677,Z 714.223,A -85,B 0,C 180,E1 9224.203,E2 9224.203} C_VEL
LIN {X 0,Y 224.389,Z 701.047,A -85,B 0,C 180,E1 9219.567,E2 9219.567} C_VEL
LIN {X 0,Y 235.307,Z 686.923,A -85,B 0,C 180,E1 9215.748,E2 9215.748} C_VEL
LIN {X 0,Y 237.558,Z 683.788,A -85,B 0,C 180,E1 9215.005,E2 9215.005} C_VEL
LIN {X 0,Y 223.558,Z 687.03,A -85,B 0,C 180,E1 9211.251,E2 9211.251} C_VEL
LIN {X 0,Y 212.078,Z 688.915,A -85,B 0,C 180,E1 9206.91,E2 9206.91} C_VEL
LIN {X 0,Y 204.402,Z 689.969,A -85,B 0,C 180,E1 9202.732,E2 9202.732} C_VEL
LIN {X 0,Y 198.502,Z 691.233,A -85,B 0,C 180,E1 9197.893,E2 9197.893} C_VEL
LIN {X 0,Y 194.157,Z 690.698,A -85,B 0,C 180,E1 9193.095,E2 9193.095} C_VEL
LIN {X 0,Y 192.414,Z 690.054,A -85,B 0,C 180,E1 9190.478,E2 9190.478} C_VEL
LIN {X 0,Y 191.225,Z 689.428,A -85,B 0,C 180,E1 9180.299,E2 9180.299} C_VEL
LIN {X 0,Y 199.871,Z 688.634,A -85,B 0,C 180,E1 9166.695,E2 9166.695} C_VEL
LIN {X 0,Y 211.65,Z 687.703,A -85,B 0,C 180,E1 9158.958,E2 9158.958} C_VEL
LIN {X 0,Y 224.533,Z 686.355,A -85,B 0,C 180,E1 9153.518,E2 9153.518} C_VEL
LIN {X 0,Y 214.369,Z 697.051,A -85,B 0,C 180,E1 9148.819,E2 9148.819} C_VEL
LIN {X 0,Y 205.265,Z 706.157,A -85,B 0,C 180,E1 9143.488,E2 9143.488} C_VEL
LIN {X 0,Y 197.672,Z 713.571,A -85,B 0,C 180,E1 9137.604,E2 9137.604} C_VEL
LIN {X 0,Y 191.942,Z 719.201,A -85,B 0,C 180,E1 9131.397,E2 9131.397} C_VEL
LIN {X 0,Y 187.943,Z 723.308,A -85,B 0,C 180,E1 9124.698,E2 9124.698} C_VEL
LIN {X 0,Y 185.743,Z 725.686,A -85,B 0,C 180,E1 9117.926,E2 9117.926} C_VEL
LIN {X 0,Y 184.908,Z 726.456,A -85,B 0,C 180,E1 9111.908,E2 9111.908} C_VEL
LIN {X 0,Y 184.707,Z 726.094,A -85,B 0,C 180,E1 9106.027,E2 9106.027} C_VEL
LIN {X 0,Y 184.877,Z 724.656,A -85,B 0,C 180,E1 9100.596,E2 9100.596} C_VEL
LIN {X 0,Y 185.763,Z 721.726,A -85,B 0,C 180,E1 9094.322,E2 9094.322} C_VEL
LIN {X 0,Y 187.764,Z 717.414,A -85,B 0,C 180,E1 9088.17,E2 9088.17} C_VEL
LIN {X 0,Y 191.325,Z 711.279,A -85,B 0,C 180,E1 9081.889,E2 9081.889} C_VEL
LIN {X 0,Y 196.778,Z 702.938,A -85,B 0,C 180,E1 9075.583,E2 9075.583} C_VEL
LIN {X 0,Y 203.625,Z 693.003,A -85,B 0,C 180,E1 9069.897,E2 9069.897} C_VEL
LIN {X 0,Y 211.565,Z 681.486,A -85,B 0,C 180,E1 9064.828,E2 9064.828} C_VEL
LIN {X 0,Y 220.268,Z 668.397,A -85,B 0,C 180,E1 9060.345,E2 9060.345} C_VEL
LIN {X 0,Y 229.47,Z 653.683,A -85,B 0,C 180,E1 9056.402,E2 9056.402} C_VEL
LIN {X 0,Y 238.616,Z 637.752,A -85,B 0,C 180,E1 9053.037,E2 9053.037} C_VEL
LIN {X 0,Y 247.464,Z 620.657,A -85,B 0,C 180,E1 9050.178,E2 9050.178} C_VEL
LIN {X 0,Y 255.787,Z 602.414,A -85,B 0,C 180,E1 9047.752,E2 9047.752} C_VEL
LIN {X 0,Y 263.1,Z 583.859,A -85,B 0,C 180,E1 9045.785,E2 9045.785} C_VEL
LIN {X 0,Y 269.567,Z 564.296,A -85,B 0,C 180,E1 9044.134,E2 9044.134} C_VEL
LIN {X 0,Y 275.12,Z 543.494,A -85,B 0,C 180,E1 9042.767,E2 9042.767} C_VEL
LIN {X 0,Y 279.485,Z 521.784,A -85,B 0,C 180,E1 9041.686,E2 9041.686} C_VEL
LIN {X 0,Y 287.019,Z 478.291,A -85,B 0,C 180,E1 9040.057,E2 9040.057} C_VEL
LIN {X 0,Y 296.92,Z 418.478,A -85,B 0,C 180,E1 9038.325,E2 9038.325} C_VEL
LIN {X 0,Y 304.005,Z 367.435,A -85,B 0,C 180,E1 9037.04,E2 9037.04} C_VEL
LIN {X 0,Y 298.017,Z 359.683,A -85,B 0,C 180,E1 9033.845,E2 9033.845} C_VEL
LIN {X 0,Y 292.296,Z 353.017,A -85,B 0,C 180,E1 9030.303,E2 9030.303} C_VEL
LIN {X 0,Y 287.794,Z 348.381,A -85,B 0,C 180,E1 9027.074,E2 9027.074} C_VEL
LIN {X 0,Y 283.93,Z 345.156,A -85,B 0,C 180,E1 9023.741,E2 9023.741} C_VEL
LIN {X 0,Y 282.394,Z 344.76,A -85,B 0,C 180,E1 9022.323,E2 9022.323} C_VEL
LIN {X 0,Y 280.035,Z 346.697,A -85,B 0,C 180,E1 9020.131,E2 9020.131} C_VEL
LIN {X 0,Y 277.67,Z 349.451,A -85,B 0,C 180,E1 9017.438,E2 9017.438} C_VEL
LIN {X 0,Y 277.165,Z 349.652,A -85,B 0,C 180,E1 9016.629,E2 9016.629} C_VEL
LIN {X 0,Y 274.877,Z 351.675,A -85,B 0,C 180,E1 9011.116,E2 9011.116} C_VEL
LIN {X 0,Y 274.617,Z 352.888,A -85,B 0,C 180,E1 9009.008,E2 9009.008} C_VEL
LIN {X 0,Y 274.683,Z 355.923,A -85,B 0,C 180,E1 9005.641,E2 9005.641} C_VEL
LIN {X 0,Y 275.704,Z 361.091,A -85,B 0,C 180,E1 9001.767,E2 9001.767} C_VEL
LIN {X 0,Y 277.976,Z 369.021,A -85,B 0,C 180,E1 8997.372,E2 8997.372} C_VEL
LIN {X 0,Y 281.042,Z 377.893,A -85,B 0,C 180,E1 8993.566,E2 8993.566} C_VEL
LIN {X 0,Y 284.182,Z 387.408,A -85,B 0,C 180,E1 8990.406,E2 8990.406} C_VEL
LIN {X 0,Y 284.53,Z 415.361,A -85,B 0,C 180,E1 8987.79,E2 8987.79} C_VEL
LIN {X 0,Y 285.488,Z 441.376,A -85,B 0,C 180,E1 8984.941,E2 8984.941} C_VEL
LIN {X 0,Y 287.212,Z 465.413,A -85,B 0,C 180,E1 8981.894,E2 8981.894} C_VEL
LIN {X 0,Y 289.17,Z 483.479,A -85,B 0,C 180,E1 8979.4,E2 8979.4} C_VEL
LIN {X 0,Y 283.511,Z 507.537,A -85,B 0,C 180,E1 8978.772,E2 8978.772} C_VEL
LIN {X 0,Y 274.762,Z 541.254,A -85,B 0,C 180,E1 8977.427,E2 8977.427} C_VEL
LIN {X 0,Y 265.654,Z 571.063,A -85,B 0,C 180,E1 8975.882,E2 8975.882} C_VEL
LIN {X 0,Y 256.774,Z 597.468,A -85,B 0,C 180,E1 8974.092,E2 8974.092} C_VEL
LIN {X 0,Y 249.362,Z 616.798,A -85,B 0,C 180,E1 8972.391,E2 8972.391} C_VEL
LIN {X 0,Y 241.167,Z 635.548,A -85,B 0,C 180,E1 8970.292,E2 8970.292} C_VEL
LIN {X 0,Y 232.433,Z 653.374,A -85,B 0,C 180,E1 8967.765,E2 8967.765} C_VEL
LIN {X 0,Y 223.267,Z 670.296,A -85,B 0,C 180,E1 8964.712,E2 8964.712} C_VEL
LIN {X 0,Y 214.241,Z 685.611,A -85,B 0,C 180,E1 8961.204,E2 8961.204} C_VEL
LIN {X 0,Y 205.187,Z 700.182,A -85,B 0,C 180,E1 8956.965,E2 8956.965} C_VEL
LIN {X 0,Y 196.94,Z 713.131,A -85,B 0,C 180,E1 8952.165,E2 8952.165} C_VEL
LIN {X 0,Y 189.548,Z 724.711,A -85,B 0,C 180,E1 8946.589,E2 8946.589} C_VEL
LIN {X 0,Y 183.647,Z 734.572,A -85,B 0,C 180,E1 8940.42,E2 8940.42} C_VEL
LIN {X 0,Y 179.598,Z 742.44,A -85,B 0,C 180,E1 8933.979,E2 8933.979} C_VEL
LIN {X 0,Y 177.325,Z 748.398,A -85,B 0,C 180,E1 8927.388,E2 8927.388} C_VEL
LIN {X 0,Y 176.551,Z 752.445,A -85,B 0,C 180,E1 8921.101,E2 8921.101} C_VEL
LIN {X 0,Y 176.631,Z 754.879,A -85,B 0,C 180,E1 8915.196,E2 8915.196} C_VEL
LIN {X 0,Y 176.76,Z 755.845,A -85,B 0,C 180,E1 8910.324,E2 8910.324} C_VEL
LIN {X 0,Y 176.578,Z 755.837,A -85,B 0,C 180,E1 8905.127,E2 8905.127} C_VEL
LIN {X 0,Y 176.432,Z 754.633,A -85,B 0,C 180,E1 8899.221,E2 8899.221} C_VEL
LIN {X 0,Y 177.323,Z 751.661,A -85,B 0,C 180,E1 8892.272,E2 8892.272} C_VEL
LIN {X 0,Y 180.146,Z 746.797,A -85,B 0,C 180,E1 8885.05,E2 8885.05} C_VEL
LIN {X 0,Y 185.236,Z 740.06,A -85,B 0,C 180,E1 8878.063,E2 8878.063} C_VEL
LIN {X 0,Y 192.336,Z 731.704,A -85,B 0,C 180,E1 8871.717,E2 8871.717} C_VEL
LIN {X 0,Y 201.807,Z 720.997,A -85,B 0,C 180,E1 8865.685,E2 8865.685} C_VEL
LIN {X 0,Y 212.24,Z 709.161,A -85,B 0,C 180,E1 8860.67,E2 8860.67} C_VEL
LIN {X 0,Y 223.531,Z 695.781,A -85,B 0,C 180,E1 8856.375,E2 8856.375} C_VEL
LIN {X 0,Y 227.939,Z 690.169,A -85,B 0,C 180,E1 8854.84,E2 8854.84} C_VEL
LIN {X 0,Y 215.061,Z 692.619,A -85,B 0,C 180,E1 8851.067,E2 8851.067} C_VEL
LIN {X 0,Y 203.351,Z 694.2,A -85,B 0,C 180,E1 8846.264,E2 8846.264} C_VEL
LIN {X 0,Y 192.069,Z 694.91,A -85,B 0,C 180,E1 8838.829,E2 8838.829} C_VEL
LIN {X 0,Y 184.512,Z 694.494,A -85,B 0,C 180,E1 8826.533,E2 8826.533} C_VEL
LIN {X 0,Y 193.662,Z 692.994,A -85,B 0,C 180,E1 8805.956,E2 8805.956} C_VEL
LIN {X 0,Y 205.759,Z 691.924,A -85,B 0,C 180,E1 8798.026,E2 8798.026} C_VEL
LIN {X 0,Y 215.751,Z 690.991,A -85,B 0,C 180,E1 8793.649,E2 8793.649} C_VEL
LIN {X 0,Y 205.108,Z 701.382,A -85,B 0,C 180,E1 8788.55,E2 8788.55} C_VEL
LIN {X 0,Y 195.802,Z 710.003,A -85,B 0,C 180,E1 8782.808,E2 8782.808} C_VEL
LIN {X 0,Y 188.028,Z 717.027,A -85,B 0,C 180,E1 8776.266,E2 8776.266} C_VEL
LIN {X 0,Y 182.472,Z 722.076,A -85,B 0,C 180,E1 8769.409,E2 8769.409} C_VEL
LIN {X 0,Y 178.901,Z 725.443,A -85,B 0,C 180,E1 8762.07,E2 8762.07} C_VEL
LIN {X 0,Y 177.313,Z 726.916,A -85,B 0,C 180,E1 8755.377,E2 8755.377} C_VEL
LIN {X 0,Y 176.78,Z 727.066,A -85,B 0,C 180,E1 8749.151,E2 8749.151} C_VEL
LIN {X 0,Y 176.779,Z 726.177,A -85,B 0,C 180,E1 8743.381,E2 8743.381} C_VEL
LIN {X 0,Y 177.289,Z 723.884,A -85,B 0,C 180,E1 8736.969,E2 8736.969} C_VEL
LIN {X 0,Y 178.897,Z 720.075,A -85,B 0,C 180,E1 8730.321,E2 8730.321} C_VEL
LIN {X 0,Y 182.029,Z 714.602,A -85,B 0,C 180,E1 8723.693,E2 8723.693} C_VEL
LIN {X 0,Y 186.558,Z 707.82,A -85,B 0,C 180,E1 8717.621,E2 8717.621} C_VEL
LIN {X 0,Y 192.966,Z 698.864,A -85,B 0,C 180,E1 8711.575,E2 8711.575} C_VEL
LIN {X 0,Y 200.567,Z 688.425,A -85,B 0,C 180,E1 8706.185,E2 8706.185} C_VEL
LIN {X 0,Y 209.057,Z 676.513,A -85,B 0,C 180,E1 8701.428,E2 8701.428} C_VEL
LIN {X 0,Y 218.634,Z 662.34,A -85,B 0,C 180,E1 8697.03,E2 8697.03} C_VEL
LIN {X 0,Y 228.04,Z 647.327,A -85,B 0,C 180,E1 8693.395,E2 8693.395} C_VEL
LIN {X 0,Y 237.514,Z 630.643,A -85,B 0,C 180,E1 8690.218,E2 8690.218} C_VEL
LIN {X 0,Y 246.226,Z 613.428,A -85,B 0,C 180,E1 8687.617,E2 8687.617} C_VEL
LIN {X 0,Y 254.291,Z 595.192,A -85,B 0,C 180,E1 8685.424,E2 8685.424} C_VEL
LIN {X 0,Y 261.564,Z 575.892,A -85,B 0,C 180,E1 8683.583,E2 8683.583} C_VEL
LIN {X 0,Y 267.919,Z 555.331,A -85,B 0,C 180,E1 8682.042,E2 8682.042} C_VEL
LIN {X 0,Y 273.118,Z 533.813,A -85,B 0,C 180,E1 8680.809,E2 8680.809} C_VEL
LIN {X 0,Y 280.445,Z 493.733,A -85,B 0,C 180,E1 8679.155,E2 8679.155} C_VEL
LIN {X 0,Y 290.656,Z 435.728,A -85,B 0,C 180,E1 8677.389,E2 8677.389} C_VEL
LIN {X 0,Y 299.155,Z 379.317,A -85,B 0,C 180,E1 8675.957,E2 8675.957} C_VEL
LIN {X 0,Y 299.96,Z 372.48,A -85,B 0,C 180,E1 8675.755,E2 8675.755} C_VEL
LIN {X 0,Y 293.979,Z 364.716,A -85,B 0,C 180,E1 8672.275,E2 8672.275} C_VEL
LIN {X 0,Y 290.13,Z 360.316,A -85,B 0,C 180,E1 8669.754,E2 8669.754} C_VEL
LIN {X 0,Y 286.194,Z 356.097,A -85,B 0,C 180,E1 8666.788,E2 8666.788} C_VEL
LIN {X 0,Y 280.166,Z 350.64,A -85,B 0,C 180,E1 8660.91,E2 8660.91} C_VEL
LIN {X 0,Y 277.165,Z 349.652,A -85,B 0,C 180,E1 8656.629,E2 8656.629} C_VEL
LIN {X 0,Y 276.301,Z 350.56,A -85,B 0,C 180,E1 8655.169,E2 8655.169} C_VEL
LIN {X 0,Y 275.034,Z 354.127,A -85,B 0,C 180,E1 8653.118,E2 8653.118} C_VEL
LIN {X 0,Y 273.761,Z 359.604,A -85,B 0,C 180,E1 8650.288,E2 8650.288} C_VEL
LIN {X 0,Y 273.627,Z 360.416,A -85,B 0,C 180,E1 8649.602,E2 8649.602} C_VEL
LIN {X 0,Y 273.592,Z 363.828,A -85,B 0,C 180,E1 8645.874,E2 8645.874} C_VEL
LIN {X 0,Y 274.46,Z 368.731,A -85,B 0,C 180,E1 8642.193,E2 8642.193} C_VEL
LIN {X 0,Y 276.63,Z 376.826,A -85,B 0,C 180,E1 8637.722,E2 8637.722} C_VEL
LIN {X 0,Y 279.427,Z 385.509,A -85,B 0,C 180,E1 8634.044,E2 8634.044} C_VEL
LIN {X 0,Y 281.651,Z 392.761,A -85,B 0,C 180,E1 8631.619,E2 8631.619} C_VEL
LIN {X 0,Y 281.617,Z 420.111,A -85,B 0,C 180,E1 8628.986,E2 8628.986} C_VEL
LIN {X 0,Y 282.13,Z 445.905,A -85,B 0,C 180,E1 8626.099,E2 8626.099} C_VEL
LIN {X 0,Y 283.404,Z 470.106,A -85,B 0,C 180,E1 8622.952,E2 8622.952} C_VEL
LIN {X 0,Y 284.745,Z 485.666,A -85,B 0,C 180,E1 8620.757,E2 8620.757} C_VEL
LIN {X 0,Y 278.889,Z 510.044,A -85,B 0,C 180,E1 8620.092,E2 8620.092} C_VEL
LIN {X 0,Y 270.868,Z 540.264,A -85,B 0,C 180,E1 8618.903,E2 8618.903} C_VEL
LIN {X 0,Y 261.565,Z 570.249,A -85,B 0,C 180,E1 8617.392,E2 8617.392} C_VEL
LIN {X 0,Y 252.719,Z 596.241,A -85,B 0,C 180,E1 8615.678,E2 8615.678} C_VEL
LIN {X 0,Y 244.852,Z 616.376,A -85,B 0,C 180,E1 8613.945,E2 8613.945} C_VEL
LIN {X 0,Y 236.047,Z 635.887,A -85,B 0,C 180,E1 8611.77,E2 8611.77} C_VEL
LIN {X 0,Y 226.944,Z 653.704,A -85,B 0,C 180,E1 8609.218,E2 8609.218} C_VEL
LIN {X 0,Y 217.377,Z 670.549,A -85,B 0,C 180,E1 8606.123,E2 8606.123} C_VEL
LIN {X 0,Y 207.888,Z 685.993,A -85,B 0,C 180,E1 8602.521,E2 8602.521} C_VEL
LIN {X 0,Y 198.485,Z 700.465,A -85,B 0,C 180,E1 8598.205,E2 8598.205} C_VEL
LIN {X 0,Y 189.787,Z 713.32,A -85,B 0,C 180,E1 8593.226,E2 8593.226} C_VEL
LIN {X 0,Y 182.154,Z 724.646,A -85,B 0,C 180,E1 8587.538,E2 8587.538} C_VEL
LIN {X 0,Y 176.229,Z 733.977,A -85,B 0,C 180,E1 8581.464,E2 8581.464} C_VEL
LIN {X 0,Y 171.883,Z 741.844,A -85,B 0,C 180,E1 8574.76,E2 8574.76} C_VEL
LIN {X 0,Y 169.423,Z 747.786,A -85,B 0,C 180,E1 8567.871,E2 8567.871} C_VEL
LIN {X 0,Y 168.563,Z 751.984,A -85,B 0,C 180,E1 8560.941,E2 8560.941} C_VEL
LIN {X 0,Y 168.661,Z 754.238,A -85,B 0,C 180,E1 8555.101,E2 8555.101} C_VEL
LIN {X 0,Y 168.793,Z 755.192,A -85,B 0,C 180,E1 8549.999,E2 8549.999} C_VEL
LIN {X 0,Y 168.57,Z 755.15,A -85,B 0,C 180,E1 8544.554,E2 8544.554} C_VEL
LIN {X 0,Y 168.479,Z 753.895,A -85,B 0,C 180,E1 8538.291,E2 8538.291} C_VEL
LIN {X 0,Y 169.609,Z 750.925,A -85,B 0,C 180,E1 8531.08,E2 8531.08} C_VEL
LIN {X 0,Y 172.879,Z 746.025,A -85,B 0,C 180,E1 8523.554,E2 8523.554} C_VEL
LIN {X 0,Y 178.539,Z 739.267,A -85,B 0,C 180,E1 8516.328,E2 8516.328} C_VEL
LIN {X 0,Y 186.628,Z 730.558,A -85,B 0,C 180,E1 8509.589,E2 8509.589} C_VEL
LIN {X 0,Y 196.461,Z 720.234,A -85,B 0,C 180,E1 8503.722,E2 8503.722} C_VEL
LIN {X 0,Y 207.534,Z 708.366,A -85,B 0,C 180,E1 8498.694,E2 8498.694} C_VEL
LIN {X 0,Y 218.444,Z 696.013,A -85,B 0,C 180,E1 8494.685,E2 8494.685} C_VEL
LIN {X 0,Y 205.538,Z 698.032,A -85,B 0,C 180,E1 8490.566,E2 8490.566} C_VEL
LIN {X 0,Y 194.667,Z 699.072,A -85,B 0,C 180,E1 8485.558,E2 8485.558} C_VEL
LIN {X 0,Y 184.283,Z 699.441,A -85,B 0,C 180,E1 8478.014,E2 8478.014} C_VEL
LIN {X 0,Y 177.733,Z 698.783,A -85,B 0,C 180,E1 8465.811,E2 8465.811} C_VEL
LIN {X 0,Y 187.366,Z 697.156,A -85,B 0,C 180,E1 8445.157,E2 8445.157} C_VEL
LIN {X 0,Y 199.846,Z 696.006,A -85,B 0,C 180,E1 8437.029,E2 8437.029} C_VEL
LIN {X 0,Y 207.027,Z 695.236,A -85,B 0,C 180,E1 8433.85,E2 8433.85} C_VEL
LIN {X 0,Y 196.573,Z 704.687,A -85,B 0,C 180,E1 8428.708,E2 8428.708} C_VEL
LIN {X 0,Y 187.202,Z 712.74,A -85,B 0,C 180,E1 8422.734,E2 8422.734} C_VEL
LIN {X 0,Y 179.344,Z 719.294,A -85,B 0,C 180,E1 8415.821,E2 8415.821} C_VEL
LIN {X 0,Y 173.778,Z 723.936,A -85,B 0,C 180,E1 8408.419,E2 8408.419} C_VEL
LIN {X 0,Y 170.576,Z 726.66,A -85,B 0,C 180,E1 8401.053,E2 8401.053} C_VEL
LIN {X 0,Y 169.173,Z 727.773,A -85,B 0,C 180,E1 8394.068,E2 8394.068} C_VEL
LIN {X 0,Y 168.772,Z 727.605,A -85,B 0,C 180,E1 8387.943,E2 8387.943} C_VEL
LIN {X 0,Y 168.859,Z 726.307,A -85,B 0,C 180,E1 8381.615,E2 8381.615} C_VEL
LIN {X 0,Y 169.64,Z 723.788,A -85,B 0,C 180,E1 8375.057,E2 8375.057} C_VEL
LIN {X 0,Y 171.778,Z 719.498,A -85,B 0,C 180,E1 8367.999,E2 8367.999} C_VEL
LIN {X 0,Y 175.568,Z 713.552,A -85,B 0,C 180,E1 8361.155,E2 8361.155} C_VEL
LIN {X 0,Y 181.133,Z 705.87,A -85,B 0,C 180,E1 8354.636,E2 8354.636} C_VEL
LIN {X 0,Y 188.063,Z 696.783,A -85,B 0,C 180,E1 8348.806,E2 8348.806} C_VEL
LIN {X 0,Y 196.461,Z 685.766,A -85,B 0,C 180,E1 8343.394,E2 8343.394} C_VEL
LIN {X 0,Y 205.689,Z 673.225,A -85,B 0,C 180,E1 8338.659,E2 8338.659} C_VEL
LIN {X 0,Y 215.424,Z 659.132,A -85,B 0,C 180,E1 8334.538,E2 8334.538} C_VEL
LIN {X 0,Y 224.774,Z 644.399,A -85,B 0,C 180,E1 8331.156,E2 8331.156} C_VEL
LIN {X 0,Y 234.383,Z 627.637,A -85,B 0,C 180,E1 8328.117,E2 8328.117} C_VEL
LIN {X 0,Y 243.137,Z 610.383,A -85,B 0,C 180,E1 8325.646,E2 8325.646} C_VEL
LIN {X 0,Y 251.496,Z 591.355,A -85,B 0,C 180,E1 8323.485,E2 8323.485} C_VEL
LIN {X 0,Y 258.663,Z 572.02,A -85,B 0,C 180,E1 8321.752,E2 8321.752} C_VEL
LIN {X 0,Y 264.867,Z 551.511,A -85,B 0,C 180,E1 8320.312,E2 8320.312} C_VEL
LIN {X 0,Y 269.858,Z 530.183,A -85,B 0,C 180,E1 8319.168,E2 8319.168} C_VEL
LIN {X 0,Y 277.698,Z 488.64,A -85,B 0,C 180,E1 8317.522,E2 8317.522} C_VEL
LIN {X 0,Y 287.837,Z 432.47,A -85,B 0,C 180,E1 8315.86,E2 8315.86} C_VEL
LIN {X 0,Y 296.158,Z 377.799,A -85,B 0,C 180,E1 8314.499,E2 8314.499} C_VEL
LIN {X 0,Y 290.822,Z 370.841,A -85,B 0,C 180,E1 8311.16,E2 8311.16} C_VEL
LIN {X 0,Y 287.575,Z 367.177,A -85,B 0,C 180,E1 8308.901,E2 8308.901} C_VEL
LIN {X 0,Y 284.329,Z 363.619,A -85,B 0,C 180,E1 8306.302,E2 8306.302} C_VEL
LIN {X 0,Y 278.921,Z 358.53,A -85,B 0,C 180,E1 8300.787,E2 8300.787} C_VEL
LIN {X 0,Y 275.774,Z 357.576,A -85,B 0,C 180,E1 8296.097,E2 8296.097} C_VEL
LIN {X 0,Y 273.627,Z 360.416,A -85,B 0,C 180,E1 8289.602,E2 8289.602} C_VEL
LIN {X 0,Y 273.364,Z 362.909,A -85,B 0,C 180,E1 8288.06,E2 8288.06} C_VEL
LIN {X 0,Y 272.915,Z 374.471,A -85,B 0,C 180,E1 8283.747,E2 8283.747} C_VEL
LIN {X 0,Y 273.125,Z 376.016,A -85,B 0,C 180,E1 8282.865,E2 8282.865} C_VEL
LIN {X 0,Y 274.93,Z 383.481,A -85,B 0,C 180,E1 8278.646,E2 8278.646} C_VEL
LIN {X 0,Y 277.45,Z 391.985,A -85,B 0,C 180,E1 8274.935,E2 8274.935} C_VEL
LIN {X 0,Y 279.212,Z 398.245,A -85,B 0,C 180,E1 8272.826,E2 8272.826} C_VEL
LIN {X 0,Y 278.72,Z 424.318,A -85,B 0,C 180,E1 8270.255,E2 8270.255} C_VEL
LIN {X 0,Y 278.777,Z 449.959,A -85,B 0,C 180,E1 8267.331,E2 8267.331} C_VEL
LIN {X 0,Y 279.626,Z 473.65,A -85,B 0,C 180,E1 8264.205,E2 8264.205} C_VEL
LIN {X 0,Y 280.499,Z 488.005,A -85,B 0,C 180,E1 8262.153,E2 8262.153} C_VEL
LIN {X 0,Y 274.491,Z 512.532,A -85,B 0,C 180,E1 8261.462,E2 8261.462} C_VEL
LIN {X 0,Y 265.558,Z 544.586,A -85,B 0,C 180,E1 8260.193,E2 8260.193} C_VEL
LIN {X 0,Y 256.84,Z 572.057,A -85,B 0,C 180,E1 8258.804,E2 8258.804} C_VEL
LIN {X 0,Y 247.55,Z 598.336,A -85,B 0,C 180,E1 8257.057,E2 8257.057} C_VEL
LIN {X 0,Y 239.754,Z 617.581,A -85,B 0,C 180,E1 8255.386,E2 8255.386} C_VEL
LIN {X 0,Y 231.087,Z 636.106,A -85,B 0,C 180,E1 8253.313,E2 8253.313} C_VEL
LIN {X 0,Y 221.348,Z 654.404,A -85,B 0,C 180,E1 8250.669,E2 8250.669} C_VEL
LIN {X 0,Y 211.149,Z 671.678,A -85,B 0,C 180,E1 8247.446,E2 8247.446} C_VEL
LIN {X 0,Y 201.047,Z 687.346,A -85,B 0,C 180,E1 8243.674,E2 8243.674} C_VEL
LIN {X 0,Y 191.164,Z 701.642,A -85,B 0,C 180,E1 8239.173,E2 8239.173} C_VEL
LIN {X 0,Y 182.18,Z 714.247,A -85,B 0,C 180,E1 8234.032,E2 8234.032} C_VEL
LIN {X 0,Y 174.439,Z 725.16,A -85,B 0,C 180,E1 8228.246,E2 8228.246} C_VEL
LIN {X 0,Y 168.205,Z 734.43,A -85,B 0,C 180,E1 8221.787,E2 8221.787} C_VEL
LIN {X 0,Y 163.844,Z 741.872,A -85,B 0,C 180,E1 8214.902,E2 8214.902} C_VEL
LIN {X 0,Y 161.286,Z 747.892,A -85,B 0,C 180,E1 8207.311,E2 8207.311} C_VEL
LIN {X 0,Y 160.566,Z 751.727,A -85,B 0,C 180,E1 8200.307,E2 8200.307} C_VEL
LIN {X 0,Y 160.722,Z 753.765,A -85,B 0,C 180,E1 8194.281,E2 8194.281} C_VEL
LIN {X 0,Y 160.79,Z 754.608,A -85,B 0,C 180,E1 8188.93,E2 8188.93} C_VEL
LIN {X 0,Y 160.549,Z 754.426,A -85,B 0,C 180,E1 8183.563,E2 8183.563} C_VEL
LIN {X 0,Y 160.598,Z 752.979,A -85,B 0,C 180,E1 8176.681,E2 8176.681} C_VEL
LIN {X 0,Y 162.33,Z 749.618,A -85,B 0,C 180,E1 8168.69,E2 8168.69} C_VEL
LIN {X 0,Y 166.428,Z 744.46,A -85,B 0,C 180,E1 8160.88,E2 8160.88} C_VEL
LIN {X 0,Y 173.238,Z 737.281,A -85,B 0,C 180,E1 8153.344,E2 8153.344} C_VEL
LIN {X 0,Y 182.207,Z 728.43,A -85,B 0,C 180,E1 8146.69,E2 8146.69} C_VEL
LIN {X 0,Y 193.015,Z 717.799,A -85,B 0,C 180,E1 8140.859,E2 8140.859} C_VEL
LIN {X 0,Y 205.639,Z 704.98,A -85,B 0,C 180,E1 8135.694,E2 8135.694} C_VEL
LIN {X 0,Y 208.751,Z 701.522,A -85,B 0,C 180,E1 8134.498,E2 8134.498} C_VEL
LIN {X 0,Y 195.441,Z 703.045,A -85,B 0,C 180,E1 8129.751,E2 8129.751} C_VEL
LIN {X 0,Y 182.085,Z 703.775,A -85,B 0,C 180,E1 8122.264,E2 8122.264} C_VEL
LIN {X 0,Y 173.711,Z 703.505,A -85,B 0,C 180,E1 8113.31,E2 8113.31} C_VEL
LIN {X 0,Y 170.898,Z 702.861,A -85,B 0,C 180,E1 8105.034,E2 8105.034} C_VEL
LIN {X 0,Y 180.596,Z 701.148,A -85,B 0,C 180,E1 8084.587,E2 8084.587} C_VEL
LIN {X 0,Y 194.456,Z 699.859,A -85,B 0,C 180,E1 8075.709,E2 8075.709} C_VEL
LIN {X 0,Y 198.069,Z 699.558,A -85,B 0,C 180,E1 8073.947,E2 8073.947} C_VEL
LIN {X 0,Y 187.302,Z 708.524,A -85,B 0,C 180,E1 8068.455,E2 8068.455} C_VEL
LIN {X 0,Y 178.095,Z 715.797,A -85,B 0,C 180,E1 8062.268,E2 8062.268} C_VEL
LIN {X 0,Y 170.537,Z 721.581,A -85,B 0,C 180,E1 8055.189,E2 8055.189} C_VEL
LIN {X 0,Y 165.232,Z 725.61,A -85,B 0,C 180,E1 8047.558,E2 8047.558} C_VEL
LIN {X 0,Y 162.276,Z 727.851,A -85,B 0,C 180,E1 8039.94,E2 8039.94} C_VEL
LIN {X 0,Y 161.087,Z 728.493,A -85,B 0,C 180,E1 8033.02,E2 8033.02} C_VEL
LIN {X 0,Y 160.778,Z 727.991,A -85,B 0,C 180,E1 8026.252,E2 8026.252} C_VEL
LIN {X 0,Y 160.992,Z 726.491,A -85,B 0,C 180,E1 8020.015,E2 8020.015} C_VEL
LIN {X 0,Y 162.143,Z 723.437,A -85,B 0,C 180,E1 8012.828,E2 8012.828} C_VEL
LIN {X 0,Y 164.875,Z 718.724,A -85,B 0,C 180,E1 8005.479,E2 8005.479} C_VEL
LIN {X 0,Y 169.676,Z 712.003,A -85,B 0,C 180,E1 7998.098,E2 7998.098} C_VEL
LIN {X 0,Y 176.179,Z 703.749,A -85,B 0,C 180,E1 7991.47,E2 7991.47} C_VEL
LIN {X 0,Y 184.447,Z 693.515,A -85,B 0,C 180,E1 7985.33,E2 7985.33} C_VEL
LIN {X 0,Y 193.817,Z 681.672,A -85,B 0,C 180,E1 7979.974,E2 7979.974} C_VEL
LIN {X 0,Y 203.922,Z 668.209,A -85,B 0,C 180,E1 7975.336,E2 7975.336} C_VEL
LIN {X 0,Y 213.811,Z 653.964,A -85,B 0,C 180,E1 7971.541,E2 7971.541} C_VEL
LIN {X 0,Y 224.087,Z 637.654,A -85,B 0,C 180,E1 7968.16,E2 7968.16} C_VEL
LIN {X 0,Y 233.92,Z 620.098,A -85,B 0,C 180,E1 7965.321,E2 7965.321} C_VEL
LIN {X 0,Y 242.743,Z 602.034,A -85,B 0,C 180,E1 7963.02,E2 7963.02} C_VEL
LIN {X 0,Y 250.745,Z 582.879,A -85,B 0,C 180,E1 7961.093,E2 7961.093} C_VEL
LIN {X 0,Y 257.793,Z 562.496,A -85,B 0,C 180,E1 7959.482,E2 7959.482} C_VEL
LIN {X 0,Y 263.465,Z 541.924,A -85,B 0,C 180,E1 7958.227,E2 7958.227} C_VEL
LIN {X 0,Y 269.495,Z 512.888,A -85,B 0,C 180,E1 7956.915,E2 7956.915} C_VEL
LIN {X 0,Y 277.668,Z 470.989,A -85,B 0,C 180,E1 7955.464,E2 7955.464} C_VEL
LIN {X 0,Y 287.483,Z 415.502,A -85,B 0,C 180,E1 7953.953,E2 7953.953} C_VEL
LIN {X 0,Y 292.4,Z 383.091,A -85,B 0,C 180,E1 7953.17,E2 7953.17} C_VEL
LIN {X 0,Y 287.189,Z 376.249,A -85,B 0,C 180,E1 7949.63,E2 7949.63} C_VEL
LIN {X 0,Y 282.677,Z 371.324,A -85,B 0,C 180,E1 7946.016,E2 7946.016} C_VEL
LIN {X 0,Y 277.62,Z 366.413,A -85,B 0,C 180,E1 7940.669,E2 7940.669} C_VEL
LIN {X 0,Y 274.635,Z 365.531,A -85,B 0,C 180,E1 7936.064,E2 7936.064} C_VEL
LIN {X 0,Y 272.541,Z 368.391,A -85,B 0,C 180,E1 7929.716,E2 7929.716} C_VEL
LIN {X 0,Y 272.469,Z 371.59,A -85,B 0,C 180,E1 7926.215,E2 7926.215} C_VEL
LIN {X 0,Y 273.125,Z 376.016,A -85,B 0,C 180,E1 7922.865,E2 7922.865} C_VEL
LIN {X 0,Y 273.481,Z 378.723,A -85,B 0,C 180,E1 7921.597,E2 7921.597} C_VEL
LIN {X 0,Y 273.767,Z 384.753,A -85,B 0,C 180,E1 7919.913,E2 7919.913} C_VEL
LIN {X 0,Y 274.342,Z 393.435,A -85,B 0,C 180,E1 7917.731,E2 7917.731} C_VEL
LIN {X 0,Y 274.886,Z 396.29,A -85,B 0,C 180,E1 7916.725,E2 7916.725} C_VEL
LIN {X 0,Y 276.805,Z 403.515,A -85,B 0,C 180,E1 7914.066,E2 7914.066} C_VEL
LIN {X 0,Y 275.91,Z 429.707,A -85,B 0,C 180,E1 7911.43,E2 7911.43} C_VEL
LIN {X 0,Y 275.533,Z 455.184,A -85,B 0,C 180,E1 7908.44,E2 7908.44} C_VEL
LIN {X 0,Y 276.007,Z 479.438,A -85,B 0,C 180,E1 7905.15,E2 7905.15} C_VEL
LIN {X 0,Y 276.373,Z 490.35,A -85,B 0,C 180,E1 7903.582,E2 7903.582} C_VEL
LIN {X 0,Y 270.06,Z 515.411,A -85,B 0,C 180,E1 7902.853,E2 7902.853} C_VEL
LIN {X 0,Y 261.247,Z 546.352,A -85,B 0,C 180,E1 7901.651,E2 7901.651} C_VEL
LIN {X 0,Y 251.017,Z 577.424,A -85,B 0,C 180,E1 7900.058,E2 7900.058} C_VEL
LIN {X 0,Y 242.403,Z 600.963,A -85,B 0,C 180,E1 7898.464,E2 7898.464} C_VEL
LIN {X 0,Y 234.447,Z 619.504,A -85,B 0,C 180,E1 7896.809,E2 7896.809} C_VEL
LIN {X 0,Y 225.537,Z 637.623,A -85,B 0,C 180,E1 7894.739,E2 7894.739} C_VEL
LIN {X 0,Y 216.261,Z 654.405,A -85,B 0,C 180,E1 7892.297,E2 7892.297} C_VEL
LIN {X 0,Y 206.544,Z 670.311,A -85,B 0,C 180,E1 7889.351,E2 7889.351} C_VEL
LIN {X 0,Y 196.179,Z 685.886,A -85,B 0,C 180,E1 7885.655,E2 7885.655} C_VEL
LIN {X 0,Y 185.95,Z 700.097,A -85,B 0,C 180,E1 7881.23,E2 7881.23} C_VEL
LIN {X 0,Y 176.403,Z 712.808,A -85,B 0,C 180,E1 7876.041,E2 7876.041} C_VEL
LIN {X 0,Y 167.932,Z 724.035,A -85,B 0,C 180,E1 7870.017,E2 7870.017} C_VEL
LIN {X 0,Y 161.28,Z 733.246,A -85,B 0,C 180,E1 7863.487,E2 7863.487} C_VEL
LIN {X 0,Y 156.364,Z 740.923,A -85,B 0,C 180,E1 7856.181,E2 7856.181} C_VEL
LIN {X 0,Y 153.56,Z 746.775,A -85,B 0,C 180,E1 7848.605,E2 7848.605} C_VEL
LIN {X 0,Y 152.601,Z 750.883,A -85,B 0,C 180,E1 7840.953,E2 7840.953} C_VEL
LIN {X 0,Y 152.74,Z 753.034,A -85,B 0,C 180,E1 7834.505,E2 7834.505} C_VEL
LIN {X 0,Y 152.83,Z 753.875,A -85,B 0,C 180,E1 7829.25,E2 7829.25} C_VEL
LIN {X 0,Y 152.572,Z 753.815,A -85,B 0,C 180,E1 7823.603,E2 7823.603} C_VEL
LIN {X 0,Y 152.634,Z 752.488,A -85,B 0,C 180,E1 7816.359,E2 7816.359} C_VEL
LIN {X 0,Y 154.391,Z 749.438,A -85,B 0,C 180,E1 7808.337,E2 7808.337} C_VEL
LIN {X 0,Y 158.959,Z 744.242,A -85,B 0,C 180,E1 7799.787,E2 7799.787} C_VEL
LIN {X 0,Y 166.205,Z 737.284,A -85,B 0,C 180,E1 7792.004,E2 7792.004} C_VEL
LIN {X 0,Y 175.753,Z 728.587,A -85,B 0,C 180,E1 7785.134,E2 7785.134} C_VEL
LIN {X 0,Y 187.107,Z 718.149,A -85,B 0,C 180,E1 7779.208,E2 7779.208} C_VEL
LIN {X 0,Y 199.197,Z 706.538,A -85,B 0,C 180,E1 7774.318,E2 7774.318} C_VEL
LIN {X 0,Y 185.154,Z 707.66,A -85,B 0,C 180,E1 7768.724,E2 7768.724} C_VEL
LIN {X 0,Y 172.408,Z 707.918,A -85,B 0,C 180,E1 7760.362,E2 7760.362} C_VEL
LIN {X 0,Y 163.993,Z 706.974,A -85,B 0,C 180,E1 7745.948,E2 7745.948} C_VEL
LIN {X 0,Y 174.151,Z 704.916,A -85,B 0,C 180,E1 7723.659,E2 7723.659} C_VEL
LIN {X 0,Y 188.478,Z 703.511,A -85,B 0,C 180,E1 7714.55,E2 7714.55} C_VEL
LIN {X 0,Y 189.187,Z 703.511,A -85,B 0,C 180,E1 7714.13,E2 7714.13} C_VEL
LIN {X 0,Y 178.392,Z 711.796,A -85,B 0,C 180,E1 7708.424,E2 7708.424} C_VEL
LIN {X 0,Y 169.081,Z 718.529,A -85,B 0,C 180,E1 7701.86,E2 7701.86} C_VEL
LIN {X 0,Y 161.915,Z 723.502,A -85,B 0,C 180,E1 7694.748,E2 7694.748} C_VEL
LIN {X 0,Y 156.79,Z 727.004,A -85,B 0,C 180,E1 7686.831,E2 7686.831} C_VEL
LIN {X 0,Y 153.983,Z 728.826,A -85,B 0,C 180,E1 7678.719,E2 7678.719} C_VEL
LIN {X 0,Y 152.979,Z 729.158,A -85,B 0,C 180,E1 7671.471,E2 7671.471} C_VEL
LIN {X 0,Y 152.809,Z 728.345,A -85,B 0,C 180,E1 7664.785,E2 7664.785} C_VEL
LIN {X 0,Y 153.223,Z 726.444,A -85,B 0,C 180,E1 7657.877,E2 7657.877} C_VEL
LIN {X 0,Y 154.844,Z 723.051,A -85,B 0,C 180,E1 7650.371,E2 7650.371} C_VEL
LIN {X 0,Y 158.272,Z 717.914,A -85,B 0,C 180,E1 7642.742,E2 7642.742} C_VEL
LIN {X 0,Y 163.947,Z 710.71,A -85,B 0,C 180,E1 7635.159,E2 7635.159} C_VEL
